# B&R Automation Studio project OpcUaSample410_BrbLibUa103 (part 2)

### RevHistory.txt
```
Revisionsgeschichte

2018-08-24	AS4.1
	Server:
		Task 'ServerData':
			-Bereitstellen von teilweisen sich ändernden Variablen über den OpcUa-Server
			-Bereistellen von Variablen, auf die die Clients schreiben können
	Client:
		Task 'ClientC' und 'ClientST':
			-Aufbauen einer Verbindung
			-Ermitteln des NamespaceIndex
			-Erzeugen von 3 Subscriptions mit MonitoredItems
			-Zyklisches Lesen einer Variablen-Liste
			-Zyklisches Schreiben einer Variablen-Liste
			-Ermitteln und Auswerten des ConnectiosStatus
			-Abbauen der Verbindung im Exit

2018-08-24	AS4.2
	Allgemein:
		-Verwendung des Rollen/Benutzer-Systems für OpcUa
		-Verwendung eines eigenen Zertifikats (Laufzeit 99 Jahre) für Server und Client
	Client:
		Task 'ClientC' und 'ClientST':
			-Hinzufügen der MonitoredItems über 'UA_MonitoredItemAddList' statt 'UA_MonitoredItemAdd'

2018-08-24	AS4.3
	Server:
		Task 'SrvMethC' und 'SrvMethST'
			-Implementierung der Methode 'Calculate'
	Client:
		Task 'ClientC' und 'ClientST':
			-Zyklischer Aufruf der Methode 'Calculate'

2018-08-24	AS4.4
	OpcUaAny:
		-Implementierung des HW-Clients, welcher nicht programmiert, sondern nur parametriert werden muss.

2018-11-19	AS4.1, AS4.2, AS4.3, AS4.4
	Client:
		Task 'ClientC' und 'ClientST':
			Das Releasen der Node-Handles, welche für die Subscription benötigt werden,
			wurde aus der Schrittkette entfernt.
			Hintergrund: Wurde die Verbindung unterbrochen und wieder hergestellt, so wurden
			die empfangenen Werte nicht mehr auf die gemappten Variablen geschrieben.
			Grundsätzlich sollten Handles nicht gelöscht werden, solange die Funktion
			benötigt wird, für die sie ermittelt wurden.

2018-11-21	AS4.4.6.71
	Server
		Task 'SrvMethC' und 'SrvMethST':
			Das ursprüngliche Projekt 'OpcUaSample44' ist aufgrund eines Fehlers in AS4.4.6.71
			nicht kompilierbar (Fehlernummer 5091), sondern nur mit AS4.4.5.61. Dehalb wurde ein
			eigenes Beispiel-Projekt 'OpcUaSample44_671' erzeugt, welches diesen Fehler umgeht.
			Hintergrund: Auf Methoden-Argumente gemappte Variablen dürfen sich in dieser Version
			nur maximal auf der 1. Ebene einer Struktur befinden, aber nicht wie im Original auf
			der 2. oder einer höheren Ebene.
			Der Fehler im AS wird schnellstmöglich (wahrscheinlich durch ein neues Upgrade)
			behoben werden.

2019-06-07	AS4.4.7.144
	Server
		Task 'SrvMethC' und 'SrvMethST':
			Der Fehler aus AS4.4.6.71 (siehe oben) wurde in dieser Version behoben. Daher wurde
			wieder auf das ursprüngliche Projekt 'OpcUaSample44' gewechselt und unter
			'OpcUaSample44_7144' abgespeichert.

2019-01-09	AS4.5
	Selbe Version wie AS4.4
		Der Fehler von '2018-11-21	AS4.4.6.71' wurde im AS behoben. Nun können auch wieder Variablen
		auf Methoden-Argumente gemappt werden, welche sich auf einer höheren Struktur-Ebene als 1 befinden.
	Überarbeitung einiger 'ReadMe.txt'-Dateien.

2019-07-05	AS4.6
	Server
		Task 'ServerData':
			Beispiele für dynamische Arrays implementiert: ByteStringExample, ByteStringExample20 und DynamicStructArray.
		Tasks 'SrvEvntC' und 'SrvEvntST':
			Beispiel zum anwenderseitigen Feuern eines Events.
		Textsystem: Sprachübersetzung des Attributs 'Description' bei den Knoten 'gVarsGlobal' und 'VarsLocal'.
	Client:
		Task 'ClientC' und 'ClientST':
			Es wurde eine Subscription implementiert, welche das Empfangen der vom Server gefeuerten Events zeigt.
	UaCerts:
		Tasks 'UaCertsC' und 'UaCertsST':
			Hier wird demonstriert, wie OpcUa-Zertifikate zur Laufzeit verwaltet werden können.

2019-07-22	AS4.6 (Eigenes Daten-Modell)
	Server
		Task 'AirCond':
			Implementierung von 3 Klima-Anlagen-Instanzen, welche über ein eigenes Modell veröffentlicht werden.
			Die Modellierung wurde komplett im externen Tool UaModeler vorgenommen.

2019-09-20	AS4.7
	AirCond (eigenes Modell):
		Es wurde ein komplett neues eigenes Modell modelliert. Die Strukturierung der Daten wurde beibehalten,
		nur deren Parametrierung wurde geändert.
		Ausserdem wurden die Vorwärts-Referenzen im externen Modell nicht mehr eingefügt. Das Mapping geschieht jetzt
		durch	Rückwärts-Referenzen, welche im AS gesetzt werden.
		Weil die Vorwärts-Referenzen auf das B&R-Modell nicht mehr nötig sind, brauchte auch das B&R-Modell nicht
		mehr ins Ua-Modeler-Projekt des eigenen Modells rückimportiert werden.
		Zusätzlich wurde ein Event 'AirConditionOperationModeChanged' implementiert. Es ist beim Knoten 'Server' und
		am Knoten der jeweiligen Instanz abgreifbar und wird immer gefeuert, wenn sich der Betriebs-Modus ändert.
	OpcUaAny:
		Durch die Verwendung eines externen Modells verschiebt sich der Namespace-Index des B&R-Modells von 6
		auf 7. Dies musste also auch in den Browse-Pfaden der OpcUaAny-Konfiguration geändert werden.
		Bei allen anderen Tasks muss nichts geändert werden, da sich diese den Namespace-Index auf das B&R-Modell
		vom Server holen.
		Leider tritt ab As4.7 + A4.73 sporadisch ein Reboot der ArSim auf, wenn im HW-Baum das Gerät 'OpcUa_any'
		aktiviert ist. Dieser Fehler ist leider noch nicht identifiziert. Daher ist das Gerät in dieser Version
		deaktiviert. Wer an dem Beispiel interessiert ist, kann das Gerät aktivieren (der Fehler tritt nicht immer
		auf). Sollte dies nicht funktionieren, kann auch mit einem älteren Beispiel gearbeitet werden, z.B. OpcUaSample46.
	ServerData:
		Das Beispiel für dynamische Arrays wurde komplett überarbeitet. Die bisherigen Beispiele wurden eliminiert und
		dafür neue implementiert, um den Unterschied zwischen 'UAArrayLength' und 'UANoOfElements' besser zu
		demonstrieren.
		Außerdem wurde die Variable 'nWritableAttributes' implementiert, um die Funktionalität 'Schreibbare Attribute'
		zu zeigen.

Hinweis zu AS4.8
	Es gibt kein Sample48, da in dieser Version keine nennenswerten neuen Funktionalitäten hinzugekommen sind.
	Es wurden nur Fehler- und Performance-Optimierungen im AS und AR gemacht.

2021-03-25	AS4.9
	Erweiterung um ein Publisher/Subscriber-Beispiel.
		Es wurde sowohl ein Publisher als auch Subscriber konfiguriert, welche zusammen passen. Auch die programmseitige
		Diagnose mittels Zähler wird demonstriert.
	Fehler in FireEvent (Task 'SrvEvent')
		Leider hat sich in der verwendeten Betriebssystem-Version A4.90 ein Fehler eingesschlichen. Wird am Field 'Context'
		eine Struktur-Variable angebunden, deren Struktur-Definition global angelegt ist (wie es legitim ist und normalerweise
		in diesem Beispiel gezeigt wird), so liefert der FB den Fehler 0x803D0000 = 'Bad_NotSupported' zurück, statt das Event zu
		feuern. Daher ist für diese Version	lediglich ein REAL angebunden. Sobald der Fehler in einer der nächsten Versionen
		behoben ist, wird das Beispiel wieder eine Struktur anbinden.

2021-09-14	As4.9 (BrbLibUa)
	Umstellung von AR A4.90 auf E4.90.
	Fehler in FireEvent (Task 'SrvEvent') ist behoben.
		Der oben beschriebene Fehler zum Field 'Context' (globale Definition der Struktur) wurde in E4.90 behoben. Daher wird hier
		auch wieder die Struktur angebunden (siehe ServerEvents\ReadMe.txt).
	Erweiterung um Bibliothek 'BrbLibUa' und deren Beispiele.
		Hier wird gezeigt, wie mithilfe dieser Bibliothek viele Funktionalitäten von Server und Client implementiert werden
		können. Im Gegensatz zur herkömmlichen Programmierung ist dann sehr viel weniger Aufwand nötig.
	Eliminierung der Hilfs-Bibliothek 'Util'
		Da alle benötigten Funktionen dieser Hilfs-Bibliothek in der Bibliothek 'BrbLib' vorhanden sind und diese sowieso
		für die 'BrbLibUa' gebraucht wird, wurde 'Util' entfernt.

2022-05-13	As4.10  (BrbLibUa V1.01)
	Umstellung von AR E4.90 auf D4.91.
	BrbLibUa V1.01 (genaueres zu Erweiterungen/Korrekturen siehe Dokumentation der Bibliothek)
	Task 'BrbUaClt': Die neue Funktion BrbUaGetSrvTimeText() wird beispielhaft verwendet.

2022-06-07	As4.10 (BrbLibUa V1.02)
	BrbLibUa V1.02 (genaueres zu Erweiterungen/Korrekturen siehe Dokumentation der Bibliothek).
	Implementierung der UnitTests für BrbLibUa.
	Die Compiler-Version wurde von V4.1.2 auf 6.3.0 geändert.
	Die Abhängigkeit von der Basis-Bibliothek 'BrbLib' wurde von V5.01 auf V5.02 geändert.
	Prüfung mit dem Code-Analyse-Tool 'ClangTidy'. Dies führt zu einer erhöhten SW-Qualität.
	Server
		Task 'SrvDt64C' und 'SrvDt64ST':
			Implementierung von 64-Bit-Datentypen wie Uint64 (ULINT) und Int64 (LINT).
	Client
		Task 'BrbUaClient': Abonnieren der Server-Info- und Server-Diagnose-Daten beispielhaft implementiert.

2024-02-22	As4.10 (BrbLibUa V1.03)
	Umstellung von AR E4.91 auf H4.91.
	Die Bibliothek BrbLib wurde von V5.02 auf V5.03 upgedatet (genaueres zu Erweiterungen/Korrekturen siehe Dokumentation der Bibliothek).
	BrbLibUa V1.03:
		Die Abhängigkeit zur Bibliothek 'BrbLib' wurde von V5.02 auf V50.3 erhöht.
		Es wurden Hinweise in die Hilfe aufgenommen.
		Die Bibliothek selbst hat sich nicht geändert.
	Prüfung mit neuer Version des Code-Analyse-Tools 'ClangTidy'. Dies führt zu einer erhöhten SW-Qualität.
	ServerEvents: Die Variable 'Fields.nSeverity' war fälschlicherweise als INT deklariert. Jetzt ist es korrekt ein UINT.
	Korrektur in den Client-Tasks 'ClientC' und 'ClientST': In folgenden Schritten wurden bei FB-Fehlermeldungen die ErrorID vom falschen
		FB übernommen: eSTEP_CREATE_SUBSCRIPT_VAR_WAIT, eSTEP_CREATE_SUBSCRIPT_EVT_WAIT.
		Dies ist jetzt korrigiert.
	ClientC und ClientST: Hinweis aufgenommen, dass zyklisches Lesen (Polling) niemals in einer Applikation implementiert werden sollte.
```

### ReadMe.txt
```
In diesem Beispiel wird die Implementierung von OpcUa-Funktionalitäten gezeigt.
Es ist KEIN offizielles Beispiel und daher besteht für den Anwender kein Anspruch auf
Erweiterung, Fehlerbehebung, Schulung oder Support. Auch die Fehlerfreiheit kann nicht
garantiert werden.

Tasks
	Template:				Ist ein Muster, um schneller neue Tasks im selben Format implementieren zu können.
									Es wird für das Beispiel nicht benötigt.
	ServerData: 		Stellt Variablen zur Verfügung, die am eigenen Server veröffentlicht werden und Variablen, welche
									von den Clients beschrieben werden.
	SrvDt64C:				Die Implementierung von 64-Bit-Werten in der Sprache ANSI-C;
	SrvDt64ST:			Die Implementierung von 64-Bit-Werten in der Sprache StructuredText;
	SrvMethC:				Die Implementierung benutzerdefinierten Server-Methoden in der Sprache ANSI-C.
	SrvMethST:			Die Implementierung benutzerdefinierten Server-Methoden in der Sprache StructuredText.
	SrvEvntC:				Anwenderseitiges Feuern eines Events in der Sprache ANSI-C.
	SrvEvntST:			Anwenderseitiges Feuern eines Events in der Sprache StructuredText. Dieser Task ist disabled.
	ClientC:				Die Implementierung des Clients in der Sprache ANSI-C.
	ClientST:				Die Implementierung des Clients in der Sprache StructuredText.
	BrbUaCltC:			Die Implementierung des Clients mithilfe der Bibiothk BrbLibUa in der Sprache ANSI-C.
	BrbUaCltST:			Die Implementierung des Clients mithilfe der Bibiothk BrbLibUa in der StructuredText.
	OpcUaAny:				Stellt lediglich Variablen bereit, welche am OpcUaAny-Client gemappt sind.
	BrbUaSrvC:			Die Implementierung des Servers mithilfe der Bibiothk BrbLibUa in der Sprache ANSI-C.
	BrbUaSrvST:			Die Implementierung des Servers mithilfe der Bibiothk BrbLibUa in der StructuredText.
	UaCertsC:				Beispiel zur Laufzeit-Verwaltung von Zertifikaten in der Sprache ANSI-C.
	UaCertsST:			Beispiel zur Laufzeit-Verwaltung von Zertifikaten in der Sprache StructuredText.
	AirCondC:				Funktionelle Implementierung für das Beispiel eines eigenen Datenmodells in der Sprache ANSI-C.
	AirCondST:			Funktionelle Implementierung für das Beispiel eines eigenen Datenmodells in der Sprache StructuredText.
	PubSub:					Exemplarische Konfiguration einer PubSub-Verbindung.

In jedem Task ist ebenfalls eine ReadMe.txt enthalten, die ihn näher beschreibt.
Der Task 'SrvEvntST' ist disabled, damit das Event nicht vom ANSIC- und vom ST-Task gefeuert wird.

Um dieses Beispiel zu verstehen, ist es zwingend notwendig, die AS-Hilfe zu studieren. Ausserdem sollte sich der
Anwender Wissen über Konzepte und die allgemeine Funktionsweise von OpcUa aneignen. B&R bietet hierfür auch Kurse an.

Ab AS4.4 kann als Ersatz für den Library-Client der OpcUa_Any-Client verwendet werden, welcher im HW-Baum
eingefügt wird und nur parametriert statt programmiert werden muss.

Ab AS4.9 kann ein Library-Client mit sehr viel weniger Aufwand mithilfe der Bibliothek BrbLibUa implementiert werden.
Auch hier ist ein Beispiel vorhanden.

WICHTIG:
Wird kein jeweils eigenes Zertifikat für Server/Client angelegt, werden beim erstmaligem Starten der SPS
automatisch Zertifikate erzeugt, welche aber nur einen Gültigkeitszeitraum von 10 Jahren haben.
Bei einer Verbindung zwischen B&R-Teilnehmern ist das unkritisch, da dann der Gültigkeitszeitraum nicht
geprüft wird. Bei einer Verbindung zu einem externen Teilnehmer (also nicht B&R) muss ermittelt werden, ob
dieser den Gültigkeitszeitraum prüft und gegebenenfalls eine Verbindugn zurückweist!
Ist das der Fall, sollten also unbedingt eigene Zertifikate angelegt und verwendet werden.
Siehe dazu AS-Hilfe GUID 'f83f9b82-60fe-4f7c-b101-504cb81ffc44' (='Access & Security/TLS/SSL(SSL bei B&R') sowie
GUID '2c919423-08bb-4895-88b8-afcf6114d0a2' (='Programmierung/Editoren/Konfigurationseditoren/
Hardwarekonfiguration/CPU Konfiguration/SG4/OPC UA Server').
In diesem Beispiel wurde jeweils ein Zertifikat für Server und Client unter
'ConfigurationView/AccessAndSecurity/CertificateStore/OwnCertifcates' mit einer Laufzeit von 50 Jahren
angelegt.
Dazu wurde die Konfiguration 'ConfigurationView/AccessAndSecurity/TransortLayerSecurity/OpcUaCfg.sslcfg'
angelegt, in welcher die Einträge konfiguriert sind.
Die Konfiguration 'SslCfgOpcUaServer' wurde dem Server in der System-Konfiguration zugewiesen.
Die Konfiguration 'SslCfgOpcUaClient' wird dem Client am FB 'UA_Connect' zugewiesen.
Siehe dazu auch Package 'UACerts'.
```

### Global.typ - Global data types
```iecst
TYPE
	OpcUaTestDatatypes_TYP : 	STRUCT
		bBool : BOOL;
		nUsint : USINT;
		nUint : UINT;
		nUdint : UDINT;
		nSint : SINT;
		nInt : INT;
		nDint : DINT;
		rReal : REAL;
		rLongReal : LREAL;
		sString : STRING[nOPCUA_STRING_CHAR_MAX];
		tTime : TIME;
		dtDateTime : DATE_AND_TIME;
		anInt : ARRAY[0..nOPCUA_ARRAY_INDEX_MAX]OF INT;
	END_STRUCT;
	OpcUaServerVars_TYP : 	STRUCT
		WriteOnly : OpcUaTestDatatypes_TYP;
		ReadOnly : OpcUaTestDatatypes_TYP;
		ReadWrite : OpcUaTestDatatypes_TYP;
	END_STRUCT;
	ClientCfgConnectionTYP : 	STRUCT
		UserIdentityToken : UAUserIdentityToken;
		tSessionTimeout : TIME;
		tMonitorConnection : TIME;
		sServerEndpointUrl : STRING[nENDPOINT_URL_CHAR_MAX];
	END_STRUCT;
	ClientCfgSubscriptionsTYP : 	STRUCT
		sNamespaceUriOrg : STRING[nNAMESPACE_URI_CHAR_MAX];
		nNamespaceUriOrg : UINT;
		sNamespaceUriBrPv : STRING[nNAMESPACE_URI_CHAR_MAX];
		nNamespaceUriBrPv : UINT;
		SubVar : ARRAY[0..nCLIENT_SUBSCRIPTION_INDEX_MAX]OF ClientCfgSubscriptionVarTYP;
		SubEvt : ClientCfgSubscriptionEvtTYP;
	END_STRUCT;
	ClientCfgSubscriptionVarTYP : 	STRUCT
		tPublishingInterval : TIME;
		nPriority : BYTE;
		MonitoredItem : ARRAY[0..nCLIENT_MONITORED_ITEM_INDEX_MAX]OF ClientCfgMonItemTYP;
	END_STRUCT;
	ClientCfgMonItemTYP : 	STRUCT
		NodeId : UANodeID;
		sVarName : STRING[nVAR_NAME_CHAR_MAX];
	END_STRUCT;
	ClientCfgSubscriptionEvtTYP : 	STRUCT
		tPublishingInterval : TIME;
		nPriority : BYTE;
		NotifierNodeId : UANodeID;
		EventTypeNodeId : UANodeID;
		EventFieldVarNames : ARRAY[0..MAX_INDEX_EVENTFIELDSELECTION]OF STRING[MAX_LENGTH_VARIABLE];
	END_STRUCT;
	ClientCfgReadTYP : 	STRUCT
		Item : ARRAY[0..nCLIENT_READ_ITEM_INDEX_MAX]OF ClientCfgMonItemTYP;
	END_STRUCT;
	ClientCfgWriteTYP : 	STRUCT
		Item : ARRAY[0..nCLIENT_WRITE_ITEM_INDEX_MAX]OF ClientCfgMonItemTYP;
	END_STRUCT;
	ClientCfgMethodsTYP : 	STRUCT
		Method : ARRAY[0..nCLIENT_METHODS_INDEX_MAX]OF ClientCfgMethodTYP;
	END_STRUCT;
	ClientCfgMethodTYP : 	STRUCT
		ObjectNodeId : UANodeID;
		MethodNodeId : UANodeID;
		ArgumentsIn : ARRAY[0..MAX_INDEX_ARGUMENTS]OF UAMethodArgument;
		ArgumentsOut : ARRAY[0..MAX_INDEX_ARGUMENTS]OF UAMethodArgument;
	END_STRUCT;
	ClientCfgTYP : 	STRUCT
		Connection : ClientCfgConnectionTYP;
		Subscriptions : ClientCfgSubscriptionsTYP;
		Read : ClientCfgReadTYP;
		Write : ClientCfgWriteTYP;
		Methods : ClientCfgMethodsTYP;
	END_STRUCT;
	ClientConnectionStatus_TYP : 	STRUCT
		eConnectionStatus : UAConnectionStatus;
		eServerState : UAServerState;
		eServerLevel : BYTE;
	END_STRUCT;
	MethCalculateArgsIn_TYP : 	STRUCT
		nVal0 : DINT;
		nVal1 : DINT;
		anArray : ARRAY[0..nMETHOD_CALC_ARRAY_INDEX_MAX]OF INT;
	END_STRUCT;
	MethCalculateArgsOut_TYP : 	STRUCT
		nAddition : DINT;
		nMultiplication : DINT;
		anArray : ARRAY[0..nMETHOD_CALC_ARRAY_INDEX_MAX]OF INT;
	END_STRUCT;
	MethCalculateArgs_TYP : 	STRUCT
		In : MethCalculateArgsIn_TYP;
		Out : MethCalculateArgsOut_TYP;
	END_STRUCT;
	EventFieldContext_TYP : 	STRUCT
		nUsint : USINT;
		rReal : REAL;
		sString : STRING[255];
	END_STRUCT;
	ClientReceivedMonItem_TYP : 	STRUCT
		bValueChanged : BOOL;
		nReceivedCount : UDINT;
	END_STRUCT;
	ProgressEvent_TYP : 	STRUCT
		nReceivedCount : UDINT;
		EventId : UAByteStringBrbEventId_TYP;
		sEventIdHex : STRING[255];
		EventType : UANodeID;
		LocalTime : UATimeZoneData;
		Message : UALocalizedText;
		ReceiveTime : UaSrv_DateTimeType;
		Severity : UINT;
		SourceName : STRING[nBRBUA_VALUE_TEXT_CHAR_MAX];
		SourceNode : UANodeID;
		Time : UaSrv_DateTimeType;
		Context : EventFieldContext_TYP;
		Progress : UINT;
	END_STRUCT;
	TransitionEvent_TYP : 	STRUCT
		nReceivedCount : UDINT;
		EventId : UAByteStringBrbEventId_TYP;
		sEventIdHex : STRING[255];
		EventType : UANodeID;
		LocalTime : UATimeZoneData;
		Message : UALocalizedText;
		ReceiveTime : UaSrv_DateTimeType;
		sReceiveTime : STRING[64];
		nSeverity : UINT;
		sSourceName : STRING[nBRBUA_VALUE_TEXT_CHAR_MAX];
		SourceNode : UANodeID;
		FromState : UALocalizedText;
		nFromStateId : UINT;
		ToState : UALocalizedText;
		nToStateId : UINT;
		Transition : UALocalizedText;
		nTransitionId : DINT;
	END_STRUCT;
	PubSubDiagDataMsg_TYP : 	STRUCT
		nTotal : UDINT;
		nError : UDINT;
	END_STRUCT;
	PubSubDiagData_TYP : 	STRUCT
		UdpMessage : PubSubDiagDataMsg_TYP;
		DataSet : PubSubDiagDataMsg_TYP;
	END_STRUCT;
END_TYPE
```

### Global.var - Global variables
```iecst
VAR CONSTANT
	nSTEP_TEXT_CHAR_MAX : UINT := 100;
	nOPCUA_STRING_CHAR_MAX : UINT := 255;
	nOPCUA_ARRAY_INDEX_MAX : UINT := 4;
	tFB_TIMEOUT : TIME := T#2s;
	nENDPOINT_URL_CHAR_MAX : UINT := 255;
	nNAMESPACE_URI_CHAR_MAX : UINT := 255;
	nCLIENT_SUBSCRIPTION_INDEX_MAX : UINT := 2;
	nCLIENT_MONITORED_ITEM_INDEX_MAX : UINT := 3;
	nCLIENT_READ_ITEM_INDEX_MAX : UINT := 2;
	nCLIENT_WRITE_ITEM_INDEX_MAX : UINT := 2;
	nCLIENT_METHODS_INDEX_MAX : UINT := 0;
	nVAR_NAME_CHAR_MAX : UINT := 255;
	nMETHOD_CALC_ARRAY_INDEX_MAX : UINT := 3;
END_VAR
```

### Package Logical/Libraries - Global libraries

### Library Logical/Libraries/BrbLib (ANSIC, version 5.03.0) - Helpful functions
Depends on: standard, astime, AsBrStr, FileIO, sys_lib, DataObj, AsUSB, AsBrWStr, ArEventLog

#### BrbLib.fun - Exported functions and function blocks
```iecst
(********************************************************************
 * COPYRIGHT -- Bernecker + Rainer
 ********************************************************************
 * Library: BrbLib
 * File: BrbLib.fun
 * Author: niedermeierr
 * Created: June 11, 2013
 ********************************************************************
 * Functions and function blocks of library BrbLib
 ********************************************************************)
(*StepHandling*)

FUNCTION BrbStepHandler : DINT (*Behandelt Schrittketten (Protokollierung, Timeout usw.)*)
	VAR_INPUT
		pStepHandling : BrbStepHandling_TYP; (*Zeiger auf eine lokale Struktur "BrbStepHandling_TYP"*)
	END_VAR
END_FUNCTION

FUNCTION BrbStartStepTimeout : UINT (*Startet den Timeout-Zähler für eine Schrittkette*)
	VAR_INPUT
		pStepHandling : BrbStepHandling_TYP; (*Zeiger auf eine lokale Struktur "BrbStepHandling_TYP"*)
		nTimeout : UDINT; (*Zeitangabe in [ms]*)
		nContinueStep : DINT; (*Schrittnummer bei abgelaufenem Timeout*)
	END_VAR
END_FUNCTION

FUNCTION BrbStopStepTimeout : UINT (*Stoppt den Timeout-Zähler für eine Schrittkette*)
	VAR_INPUT
		pStepHandling : BrbStepHandling_TYP; (*Zeiger auf eine lokale Struktur "BrbStepHandling_TYP"*)
	END_VAR
END_FUNCTION

FUNCTION BrbStartStopWatch : BOOL (*Startet eine Stoppuhr*)
	VAR_INPUT
		pStopWatch : BrbStopWatch_TYP; (*Zeiger auf eine lokale Struktur "BrbStopWatch_TYP"*)
	END_VAR
END_FUNCTION

FUNCTION BrbStopStopWatch : UDINT (*Stoppt eine Stoppuhr*)
	VAR_INPUT
		pStopWatch : BrbStopWatch_TYP; (*Zeiger auf eine lokale Struktur "BrbStopWatch_TYP"*)
	END_VAR
END_FUNCTION
(*TaskCommunication*)

FUNCTION BrbSetCaller : BrbCallerStates_ENUM (*Versucht, die Reservierung für ein Task-Kommando zu erhalten*)
	VAR_INPUT
		pCaller : BrbCaller_TYP; (*Zeiger auf eine Struktur "BrbCaller_TYP"*)
		nCallerId : DINT; (*Identifier für den aufrufenden Task*)
	END_VAR
END_FUNCTION

FUNCTION BrbClearDirectBox : UINT (*Setzt eine DirectBox komplett auf 0*)
	VAR_INPUT
		pDirectBox : UDINT; (*Zeiger auf eine DirectBox-Struktur*)
		nSize : UDINT; (*Größe der Struktur*)
	END_VAR
END_FUNCTION

FUNCTION BrbClearCallerBox : UINT (*Setzt eine CallerBox komplett auf 0*)
	VAR_INPUT
		pCallerBox : UDINT; (*Zeiger auf eine CallerBox-Struktur*)
		nSize : UDINT; (*Größe der Struktur*)
	END_VAR
END_FUNCTION
(*VarHandling*)

{REDUND_UNREPLICABLE} FUNCTION_BLOCK BrbSaveVarAscii (*Speichert eine Variable mit allen Elementen in einer Ascii-Datei*)
	VAR_INPUT
		pDevice : REFERENCE TO STRING[0]; (*Zeiger auf den Laufwerks-Namen*)
		pFile : REFERENCE TO STRING[0]; (*Zeiger auf den Datei-Namen*)
		pVarName : REFERENCE TO STRING[0]; (*Zeiger auf den Variablen-Namen*)
		nLinesToWriteAtOneStep : {REDUND_UNREPLICABLE} UINT; (*Anzahl der Zeilen, die in einem Aufruf geschrieben werden*)
	END_VAR
	VAR_OUTPUT
		nCharCountMaxPerWrite : {REDUND_UNREPLICABLE} UDINT; (*Größte Anzahl der Zeichen, welche in einer Zeile geschrieben wurden*)
		nStatus : {REDUND_UNREPLICABLE} UINT; (*Fub-Status*)
	END_VAR
	VAR
		eStep : {REDUND_UNREPLICABLE} DINT; (*Step-Nummer für die interne Schrittkette*)
		nStatusIntern : {REDUND_UNREPLICABLE} UINT; (*Interner Fub-Status*)
		fbFileDelete : {REDUND_UNREPLICABLE} FileDelete; (*Fub zum Löschen der Datei*)
		fbFileCreate : {REDUND_UNREPLICABLE} FileCreate; (*Fub zum Erzeugen der Datei*)
		sHelp : {REDUND_UNREPLICABLE} STRING[nBRB_PVNAME_CHAR_MAX]; (*Hilfsstring*)
		nOffset : {REDUND_UNREPLICABLE} UDINT; (*Schreib-Offset*)
		nLineCountWrite : {REDUND_UNREPLICABLE} UDINT; (*Zeilen-Zähler*)
		bVarFinished : {REDUND_UNREPLICABLE} BOOL; (*1= Variable komplett durchgetickert*)
		PvInfo : {REDUND_UNREPLICABLE} ARRAY[0..16] OF BrbPvInfo_TYP; (*Struktur für Variablen-Daten*)
		nPvLevel : {REDUND_UNREPLICABLE} UINT; (*Hierarchie-Level für Strukturen*)
		sLines : {REDUND_UNREPLICABLE} STRING[nBRB_FILE_LINES_CHAR_MAX]; (*Text-Zeilen*)
		fbFileWrite : {REDUND_UNREPLICABLE} FileWrite; (*Fub zum Schreiben der Datei*)
		fbFileClose : {REDUND_UNREPLICABLE} FileClose; (*Fub zum Schliessen der Datei*)
	END_VAR
END_FUNCTION_BLOCK

FUNCTION_BLOCK BrbLoadVarAscii (*Lädt eine Ascii-Datei mit Variablen-Werten*)
	VAR_INPUT
		pDevice : REFERENCE TO STRING[0]; (*Zeiger auf den Laufwerks-Namen*)
		pFile : REFERENCE TO STRING[0]; (*Zeiger auf den Datei-Namen*)
		eLineBeak : BrbLineBreak_ENUM; (*Verwendeter Zeilenumbruch*)
		nLinesToReadAtOneStep : {REDUND_UNREPLICABLE} UINT; (*Anzahl der Zeilen, die in einem Aufruf gelesen werden*)
	END_VAR
	VAR_OUTPUT
		nStatus : {REDUND_UNREPLICABLE} UINT; (*Fub-Status*)
	END_VAR
	VAR
		eStep : {REDUND_UNREPLICABLE} DINT; (*Step-Nummer für die interne Schrittkette*)
		nStatusIntern : {REDUND_UNREPLICABLE} UINT; (*Interner Fub-Status*)
		fbDatObjInfo : {REDUND_UNREPLICABLE} DatObjInfo; (*Fub zum Holen der Datenobjekt-Info*)
		fbFileOpen : {REDUND_UNREPLICABLE} FileOpen; (*Fub zum Öffnen der Datei*)
		fbDatObjCreate : {REDUND_UNREPLICABLE} DatObjCreate; (*Fub zum Erzeugen des Datenobjekts*)
		sLineBreak : STRING[8]; (*Verwendeter Zeilenumbruch*)
		pTextStart : REFERENCE TO STRING[0]; (*Zeiger auf den Anfang des eingelesenen Texts*)
		pTextEnd : REFERENCE TO STRING[0]; (*Zeiger auf das Ende des eingelesenen Texts*)
		pText : REFERENCE TO STRING[0]; (*Zeiger auf den aktuellen Text*)
		nLineCountRead : {REDUND_UNREPLICABLE} UDINT; (*Anzahl der eingelesenen Zeilen*)
		fbFileRead : {REDUND_UNREPLICABLE} FileRead; (*Fub zum Lesen der Datei*)
		fbFileClose : {REDUND_UNREPLICABLE} FileClose; (*Fub zum Schliessen der Datei*)
		fbDatObjDelete : {REDUND_UNREPLICABLE} DatObjDelete; (*Fub zum Löschen des Datenobjekts*)
	END_VAR
END_FUNCTION_BLOCK

{REDUND_UNREPLICABLE} FUNCTION_BLOCK BrbSaveVarBin (*Speichert eine Variable mit allen Elementen in einer Binär-Datei*)
	VAR_INPUT
		pDevice : REFERENCE TO STRING[0]; (*Zeiger auf den Laufwerks-Namen*)
		pFile : REFERENCE TO STRING[0]; (*Zeiger auf den Datei-Namen*)
		pVarName : REFERENCE TO STRING[0]; (*Zeiger auf den Variablen-Namen*)
	END_VAR
	VAR_OUTPUT
		nStatus : {REDUND_UNREPLICABLE} UINT; (*Fub-Status*)
	END_VAR
	VAR
		eStep : {REDUND_UNREPLICABLE} DINT; (*Step-Nummer für die interne Schrittkette*)
		nStatusIntern : {REDUND_UNREPLICABLE} UINT; (*Interner Fub-Status*)
		PvInfo : {REDUND_UNREPLICABLE} BrbPvInfo_TYP; (*Struktur für Variablen-Daten*)
		fbFileDelete : {REDUND_UNREPLICABLE} FileDelete; (*Fub zum Löschen der Datei*)
		fbFileCreate : {REDUND_UNREPLICABLE} FileCreate; (*Fub zum Erzeugen der Datei*)
		fbFileWrite : {REDUND_UNREPLICABLE} FileWrite; (*Fub zum Schreiben der Datei*)
		fbFileClose : {REDUND_UNREPLICABLE} FileClose; (*Fub zum Schliessen der Datei*)
	END_VAR
END_FUNCTION_BLOCK

{REDUND_UNREPLICABLE} FUNCTION_BLOCK BrbLoadVarBin (*Lädt eine Binär-Datei mit Variablen-Werten*)
	VAR_INPUT
		pDevice : REFERENCE TO STRING[0]; (*Zeiger auf den Laufwerks-Namen*)
		pFile : REFERENCE TO STRING[0]; (*Zeiger auf den Datei-Namen*)
		pVarName : REFERENCE TO STRING[0]; (*Zeiger auf den Variablen-Namen*)
		bAllowBiggerVar : {REDUND_UNREPLICABLE} BOOL; (*1=Der Speicher der Variablen darf größer als die Datei sein*)
	END_VAR
	VAR_OUTPUT
		nStatus : {REDUND_UNREPLICABLE} UINT; (*Fub-Status*)
	END_VAR
	VAR
		eStep : {REDUND_UNREPLICABLE} DINT; (*Step-Nummer für die interne Schrittkette*)
		nStatusIntern : {REDUND_UNREPLICABLE} UINT; (*Interner Fub-Status*)
		fbFileOpen : {REDUND_UNREPLICABLE} FileOpen; (*Fub zum Öffnen der Datei*)
		PvInfo : {REDUND_UNREPLICABLE} BrbPvInfo_TYP; (*Struktur für Variablen-Daten*)
		fbFileRead : {REDUND_UNREPLICABLE} FileRead; (*Fub zum Lesen der Datei*)
		fbFileClose : {REDUND_UNREPLICABLE} FileClose; (*Fub zum Schliessen der Datei*)
	END_VAR
END_FUNCTION_BLOCK
(*FileHandling*)

{REDUND_UNREPLICABLE} FUNCTION_BLOCK BrbReadDir (*Gibt eine Liste der Dateien und/oder der Verzeichnisse eines Laufwerks zurück*)
	VAR_INPUT
		pDevice : REFERENCE TO STRING[0]; (*Zeiger auf den Laufwerks-Namen*)
		pPath : REFERENCE TO STRING[0]; (*Zeiger auf den Pfad*)
		eFilter : {REDUND_UNREPLICABLE} BrbDirInfoFilter_ENUM; (*Datei- und Verzeichnis-Filter*)
		bWithParentDir : {REDUND_UNREPLICABLE} BOOL; (*1=Mit übergeordnetem Verzeichnis*)
		pFileFilter : REFERENCE TO STRING[0]; (*Zeiger auf den Filtertext für Datei-Endungen*)
		bUserFilter : {REDUND_UNREPLICABLE} BOOL; (*1=Benutzerdefinierte Filterfunktion wird zusätzlich verwendet*)
		pUserFilterFunction : {REDUND_UNREPLICABLE} UDINT; (*Zeiger auf die benutzerdefinierte Filterfunktion*)
		eSorting : {REDUND_UNREPLICABLE} BrbFileSorting_ENUM; (*Sortierung*)
		bCaseSensitive : {REDUND_UNREPLICABLE} BOOL; (*1=Groß-/Klein-Schreibung beachten (gitl nur bei alphanumerischer Sortierung)*)
		pUserCompareFunction : {REDUND_UNREPLICABLE} UDINT; (*Zeiger auf die benutzerdefinierte Vergleichsfunktion bei 'eBRB_FILE_SORTING_USER'*)
		pList : {REDUND_UNREPLICABLE} UDINT; (*Zeiger auf das zu füllende Array*)
		nListIndexMax : {REDUND_UNREPLICABLE} UDINT; (*Maximaler Anzahl der Einträge im Array*)
	END_VAR
	VAR_OUTPUT
		nDirCount : {REDUND_UNREPLICABLE} UDINT; (*Anzahl der Verzeichnisse in der Liste*)
		nFileCount : {REDUND_UNREPLICABLE} UDINT; (*Anzahl der Dateien in der Liste*)
		nTotalCount : {REDUND_UNREPLICABLE} UDINT; (*Anzahl der Verzeichnisse und Dateien in der Liste*)
		nStatus : {REDUND_UNREPLICABLE} UINT; (*Fub-Status*)
	END_VAR
	VAR
		eStep : {REDUND_UNREPLICABLE} DINT; (*Step-Nummer für die interne Schrittkette*)
		FilterListMan : {REDUND_UNREPLICABLE} BrbMemListManagement_Typ; (*Verwaltung der Filter-Liste*)
		FilterList : {REDUND_UNREPLICABLE} ARRAY[0..nBRB_FILTER_SINGLE_INDEX_MAX] OF STRING[nBRB_FILTER_SINGLE_CHAR_MAX]; (*Liste der Filter*)
		fbDirRead : {REDUND_UNREPLICABLE} DirRead; (*Fub zum Auslesen des Laufwerks*)
		FileInfo : {REDUND_UNREPLICABLE} fiDIR_READ_DATA; (*Daten der aktueller Datei*)
		ReadListEntry : {REDUND_UNREPLICABLE} BrbReadDirListEntry_TYP; (*Daten der aktueller Datei*)
		FileListMan : {REDUND_UNREPLICABLE} BrbMemListManagement_Typ; (*Verwaltung der Datei-Liste*)
	END_VAR
END_FUNCTION_BLOCK

{REDUND_UNREPLICABLE} FUNCTION_BLOCK BrbCheckUsbSticks (*Prüft, ob ein Usb-Stick gesteckt wurde*)
	VAR_INPUT
		bAutoLink : {REDUND_UNREPLICABLE} BOOL; (*1=Usb-Device wird beim Stecken automatisch gelinkt*)
	END_VAR
	VAR_OUTPUT
		nUsbDeviceCount : {REDUND_UNREPLICABLE} UINT; (*Anzahl der gesteckten Usb-Sticks*)
		bUsbDeviceCountChanged : {REDUND_UNREPLICABLE} BOOL; (*Anzahl hat sich geändert (nur 1 für einen Zyklus)*)
		UsbDeviceList : {REDUND_UNREPLICABLE} ARRAY[0..nBRB_USB_DEVICE_LIST_INDEX_MAX] OF BrbUsbDeviceListEntry_TYP; (*Liste der Usb-Devices*)
		nStatus : {REDUND_UNREPLICABLE} UINT; (*Fub-Status*)
	END_VAR
	VAR
		eStep : {REDUND_UNREPLICABLE} DINT; (*Step-Nummer für die interne Schrittkette*)
		DeviceListMan : {REDUND_UNREPLICABLE} BrbMemListManagement_Typ; (*Verwaltung der Device-Liste*)
		nUsbDeviceIndex : {REDUND_UNREPLICABLE} UINT; (*Aktueller Index in der Device-Liste*)
		UsbDeviceListEntry : {REDUND_UNREPLICABLE} BrbUsbDeviceListEntry_TYP; (*Aktueller Eintrag in der Device-Liste*)
		fbUsbNodeListGet : {REDUND_UNREPLICABLE} UsbNodeListGet; (*Fub zum Lesen der Node-Liste*)
		nUsbNodeIndex : {REDUND_UNREPLICABLE} UINT; (*Aktueller Index in der Node-Liste*)
		UsbNodeList : {REDUND_UNREPLICABLE} ARRAY[0..nBRB_USB_DEVICE_LIST_INDEX_MAX] OF UDINT; (*Node-Liste*)
		nAttachDetachCountOld : {REDUND_UNREPLICABLE} UDINT; (*Vergleichs-Zähler*)
		fbDevUnlink : {REDUND_UNREPLICABLE} DevUnlink; (*Fub zum Unlinken*)
		fbUsbNodeGet : {REDUND_UNREPLICABLE} UsbNodeGet; (*Fub zum Lesen der Node-Info*)
		UsbNodeInfo : {REDUND_UNREPLICABLE} usbNode_typ; (*Node-Info*)
		sLinkParameter : {REDUND_UNREPLICABLE} STRING[100]; (*Parameter zum Linken*)
		fbDevLink : {REDUND_UNREPLICABLE} DevLink; (*Fub zum Linken*)
	END_VAR
END_FUNCTION_BLOCK

{REDUND_UNREPLICABLE} FUNCTION_BLOCK BrbDeleteFiles (*Löscht Dateien, die über Filter festgelegt sind*)
	VAR_INPUT
		pDevice : REFERENCE TO STRING[0]; (*Zeiger auf den Laufwerks-Namen*)
		pPath : REFERENCE TO STRING[0]; (*Zeiger auf den Pfad*)
		pFileFilter : REFERENCE TO STRING[0]; (*Zeiger auf den Filtertext für Datei-Endungen*)
		dtDateStart : {REDUND_UNREPLICABLE} DATE_AND_TIME; (*Angabe des Start-Datums*)
		dtDateEnd : {REDUND_UNREPLICABLE} DATE_AND_TIME; (*Angabe des Ende-Datums*)
	END_VAR
	VAR_OUTPUT
		nDeletedFileCount : {REDUND_UNREPLICABLE} UDINT; (*Anzahl der gelöschten Dateien*)
		nKeptFileCount : {REDUND_UNREPLICABLE} UDINT; (*Anzahl der nicht gelöschten Dateien*)
		nStatus : {REDUND_UNREPLICABLE} UINT; (*Fub-Status*)
	END_VAR
	VAR
		eStep : {REDUND_UNREPLICABLE} DINT; (*Step-Nummer für die interne Schrittkette*)
		FilterListMan : {REDUND_UNREPLICABLE} BrbMemListManagement_Typ; (*Verwaltung der Filter-Liste*)
		FilterList : {REDUND_UNREPLICABLE} ARRAY[0..nBRB_FILTER_SINGLE_INDEX_MAX] OF STRING[nBRB_FILTER_SINGLE_CHAR_MAX]; (*Liste der Filter*)
		fbDirRead : {REDUND_UNREPLICABLE} DirRead; (*Fub zum Auslesen des Laufwerks*)
		FileInfo : {REDUND_UNREPLICABLE} fiDIR_READ_DATA; (*Daten der aktueller Datei*)
		sFileWithPath : {REDUND_UNREPLICABLE} STRING[nBRB_FILE_NAME_CHAR_MAX]; (*Pfad mit Dateiname*)
		fbFileDelete : {REDUND_UNREPLICABLE} FileDelete; (*Fub zum Auslesen des Laufwerks*)
	END_VAR
END_FUNCTION_BLOCK

{REDUND_UNREPLICABLE} FUNCTION_BLOCK BrbLoadFileDataObj (*Lädt eine Datei in ein Datenobjekt*)
	VAR_INPUT
		pDevice : REFERENCE TO STRING[0]; (*Zeiger auf den Laufwerks-Namen*)
		pFile : REFERENCE TO STRING[0]; (*Zeiger auf den Datei-Namen*)
		pDataObjName : REFERENCE TO STRING[0]; (*Zeiger auf den Datenobjekt-Namen*)
		nDataObjMemType : {REDUND_UNREPLICABLE} USINT; (*Angabe über den Speicher-Typ des Datenobjekts*)
		nDataObjOption : {REDUND_UNREPLICABLE} UDINT; (*Angabe über die Option des Datenobjekts*)
	END_VAR
	VAR_OUTPUT
		nStatus : {REDUND_UNREPLICABLE} UINT; (*Fub-Status*)
		nDataObjIdent : {REDUND_UNREPLICABLE} UDINT; (*Ident des Datenobjekts*)
		pDataObjMem : {REDUND_UNREPLICABLE} UDINT; (*Zeiger auf die Daten des Datenobjekts*)
		nDataObjLen : {REDUND_UNREPLICABLE} UDINT; (*Länge des Datenobjekts (= Länge der Datei)*)
	END_VAR
	VAR
		eStep : {REDUND_UNREPLICABLE} DINT; (*Step-Nummer für die interne Schrittkette*)
		nStatusIntern : {REDUND_UNREPLICABLE} UINT; (*Interner Fub-Status*)
		fbDatObjInfo : {REDUND_UNREPLICABLE} DatObjInfo; (*Interner Fub*)
		fbDatObjDelete : {REDUND_UNREPLICABLE} DatObjDelete; (*Interner Fub*)
		fbFileOpen : {REDUND_UNREPLICABLE} FileOpen; (*Interner Fub*)
		fbDatObjCreate : {REDUND_UNREPLICABLE} DatObjCreate; (*Interner Fub*)
		fbFileRead : {REDUND_UNREPLICABLE} FileRead; (*Interner Fub*)
		fbFileClose : {REDUND_UNREPLICABLE} FileClose; (*Interner Fub*)
	END_VAR
END_FUNCTION_BLOCK

{REDUND_UNREPLICABLE} FUNCTION_BLOCK BrbSaveFileDataObj (*Speichert ein Datenobjekt in eine Datei*)
	VAR_INPUT
		pDevice : REFERENCE TO STRING[0]; (*Zeiger auf den Laufwerks-Namen*)
		pFile : REFERENCE TO STRING[0]; (*Zeiger auf den Datei-Namen*)
		pDataObjName : REFERENCE TO STRING[0]; (*Zeiger auf den Datenobjekt-Namen*)
	END_VAR
	VAR_OUTPUT
		nStatus : {REDUND_UNREPLICABLE} UINT; (*Fub-Status*)
	END_VAR
	VAR
		eStep : {REDUND_UNREPLICABLE} DINT; (*Step-Nummer für die interne Schrittkette*)
		nStatusIntern : {REDUND_UNREPLICABLE} UINT; (*Interner Fub-Status*)
		fbDatObjInfo : {REDUND_UNREPLICABLE} DatObjInfo; (*Interner Fub*)
		fbFileInfo : {REDUND_UNREPLICABLE} FileInfo; (*Interner Fub*)
		FileInfo : {REDUND_UNREPLICABLE} fiFILE_INFO; (*Interne Daten*)
		fbFileDelete : {REDUND_UNREPLICABLE} FileDelete; (*Interner Fub*)
		fbFileCreate : {REDUND_UNREPLICABLE} FileCreate; (*Interner Fub*)
		fbFileWrite : {REDUND_UNREPLICABLE} FileWrite; (*Interner Fub*)
		fbFileClose : {REDUND_UNREPLICABLE} FileClose; (*Interner Fub*)
	END_VAR
END_FUNCTION_BLOCK

{REDUND_UNREPLICABLE} FUNCTION_BLOCK BrbLoadFileBin (*Lädt eine Datei in eine Feld-Variable*) (*$GROUP=User,$CAT=User,$GROUPICON=User.png,$CATICON=User.png*)
	VAR_INPUT
		pDevice : REFERENCE TO STRING[0]; (*Zeiger auf den Laufwerks-Namen*)
		pFile : REFERENCE TO STRING[0]; (*Zeiger auf den Datei-Namen*)
		pVar : REFERENCE TO USINT; (*Zeiger auf die Feld-Variable*)
		nVarSize : {REDUND_UNREPLICABLE} UDINT; (*Größe der Feld-Variable*)
	END_VAR
	VAR_OUTPUT
		nStatus : {REDUND_UNREPLICABLE} UINT; (*Fub-Status*)
		nValidBytes : {REDUND_UNREPLICABLE} UDINT; (*Anzahl der gelesenen Bytes*)
	END_VAR
	VAR
		eStep : {REDUND_UNREPLICABLE} DINT; (*Step-Nummer für die interne Schrittkette*)
		nStatusIntern : {REDUND_UNREPLICABLE} UINT; (*Interner Fub-Status*)
		fbFileOpen : {REDUND_UNREPLICABLE} FileOpen; (*Interner Fub*)
		fbFileReadEx : {REDUND_UNREPLICABLE} FileReadEx; (*Interner Fub*)
		fbFileClose : {REDUND_UNREPLICABLE} FileClose; (*Interner Fub*)
	END_VAR
END_FUNCTION_BLOCK

FUNCTION BrbCheckFileName : UINT (*Ersetzt Sonderzeichen in einem Datei-Namen mit Unterstrichen*)
	VAR_INPUT
		pFileName : STRING[0]; (*Zeiger auf den Datei-Namen*)
	END_VAR
END_FUNCTION

FUNCTION BrbCheckFileEnding : BOOL (*Prüft die Endung eines Datei-Namens und berichtigt sie gegebenenfalls*)
	VAR_INPUT
		pFileName : STRING[0]; (*Zeiger auf den Datei-Namen*)
		pEnding : STRING[0]; (*Zeiger auf die Datei-Endung (mit oder ohne Punkt)*)
	END_VAR
END_FUNCTION

FUNCTION BrbCombinePath : UINT (*Fügt zwei Pfade oder einen Pfad und eine Datei-Namen zusammen*)
	VAR_INPUT
		pPath : STRING[0]; (*Zeiger auf Pfad*)
		pFilename : STRING[0]; (*Zeiger auf Pfad oder Datei-Namen*)
		pFilenameWithPath : STRING[0]; (*Zeiger auf den String, der das Ergebnis aufnimmt*)
	END_VAR
END_FUNCTION
(*Logger*)

{REDUND_UNREPLICABLE} FUNCTION_BLOCK BrbLoggerReadHierarchicalList (*Liest die zu einem definierten Logger-Eintrag gehörende Hierarchie-Liste von Einträgen aus*) (*$GROUP=User,$CAT=User,$GROUPICON=User.png,$CATICON=User.png*)
	VAR_INPUT
		sLogbookName : {REDUND_UNREPLICABLE} STRING[256]; (*Name des Logbuchs*)
		nStartRecordId : {REDUND_UNREPLICABLE} ArEventLogRecordIDType; (*RecordId, bei dem die Suche beginnen soll (0=Beginn bei jüngstem Eintrag)*)
		sObjectId : {REDUND_UNREPLICABLE} STRING[36]; (*ObjectId-Filter ('Entered by'-Angabe)*)
		nStartEventId : {REDUND_UNREPLICABLE} DINT; (*EventId oder ErrorNumber, bei dem die Liste beginnen soll (0=keine Filterung)*)
		eSeverities : {REDUND_UNREPLICABLE} BrbLogHierarchListSevFilter_ENUM; (*Bitweise codierte Filterung der Severities (0=keine Filterung)*)
		sLanguageCode : {REDUND_UNREPLICABLE} ArEventLogLanguageCodeType; (*Sprachkürzel*)
		nSearchEntryCountLimit : {REDUND_UNREPLICABLE} UDINT; (*Limitierung der durchsuchten Einträge (0=kein Limit)*)
		pLogList : {REDUND_UNREPLICABLE} UDINT; (*Zeiger auf die zu füllende Liste*)
		nLogListIndexMax : {REDUND_UNREPLICABLE} UINT; (*Maximaler Index der Liste*)
	END_VAR
	VAR_OUTPUT
		nListEntryCount : {REDUND_UNREPLICABLE} UINT; (*Anzahl der Einträge in der Liste*)
		nStatus : {REDUND_UNREPLICABLE} DINT; (*Fub-Status*)
	END_VAR
	VAR
		eStep : {REDUND_UNREPLICABLE} DINT; (*Step-Nummer für die interne Schrittkette*)
		sLastLogbookName : {REDUND_UNREPLICABLE} STRING[256]; (*Name des Logbuchs beim letzten Aufruf*)
		fbArEventLogGetIdent : {REDUND_UNREPLICABLE} ArEventLogGetIdent; (*Interner Fub*)
		nEventLogIdent : {REDUND_UNREPLICABLE} ArEventLogIdentType; (*Ident des Logbuchs*)
		ActEntry : {REDUND_UNREPLICABLE} BrbLogHierarchListEntry_TYP; (*Aktuell ermittelter Eintrag*)
		fbArEventLogGetLatestRecordID : {REDUND_UNREPLICABLE} ArEventLogGetLatestRecordID; (*Interner Fub*)
		fbArEventLogGetPreviousRecordID : {REDUND_UNREPLICABLE} ArEventLogGetPreviousRecordID; (*Interner Fub*)
		fbArEventLogRead : {REDUND_UNREPLICABLE} ArEventLogRead; (*Interner Fub*)
		fbArEventLogReadErrorNumber : {REDUND_UNREPLICABLE} ArEventLogReadErrorNumber; (*Interner Fub*)
		fbArEventLogReadObjectID : {REDUND_UNREPLICABLE} ArEventLogReadObjectID; (*Interner Fub*)
		fbArEventLogReadDescription : {REDUND_UNREPLICABLE} ArEventLogReadDescription; (*Interner Fub*)
		LogListManagement : {REDUND_UNREPLICABLE} BrbMemListManagement_Typ; (*Verwaltung der Liste*)
		nSearchEntryCount : {REDUND_UNREPLICABLE} UDINT; (*Anzahl der durchsuchten Einträge*)
		bFirstEntryIsListed : {REDUND_UNREPLICABLE} BOOL; (*Erster Eintrag lt. Filter eingetragen*)
	END_VAR
END_FUNCTION_BLOCK
(*TimeAndDate*)

FUNCTION BrbSetDtStruct : DATE_AND_TIME (*Setzt eine DTStructure-Zeit*) (*$GROUP=User,$CAT=User,$GROUPICON=User.png,$CATICON=User.png*)
	VAR_INPUT
		pDtStruct : DTStructure; (*Zeiger auf eine Zeit-Struktur*)
		nYear : UINT; (*Jahr*)
		nMonth : USINT; (*Monat*)
		nDay : USINT; (*Tage*)
		nHour : USINT; (*Stunde*)
		nMinute : USINT; (*Minute*)
		nSecond : USINT; (*Sekunde*)
		nMillisecond : UINT; (*Millisekunde*)
		nMicrosecond : UINT; (*Mikrosekunden*)
	END_VAR
END_FUNCTION

FUNCTION BrbSetDt : DATE_AND_TIME (*Setzt eine DATE_AND_TIME-Zeit*) (*$GROUP=User,$CAT=User,$GROUPICON=User.png,$CATICON=User.png*)
	VAR_INPUT
		nYear : UINT; (*Jahr*)
		nMonth : USINT; (*Monat*)
		nDay : USINT; (*Tage*)
		nHour : USINT; (*Stunde*)
		nMinute : USINT; (*Minute*)
		nSecond : USINT; (*Sekunde*)
	END_VAR
END_FUNCTION

FUNCTION BrbSetTimespan : TIME (*Setzt eine TIME-Zeitspanne*) (*$GROUP=User,$CAT=User,$GROUPICON=User.png,$CATICON=User.png*)
	VAR_INPUT
		nSign : SINT; (*Vorzeichen*)
		nDays : UDINT; (*Tage*)
		nHours : UDINT; (*Stunden*)
		nMinutes : UDINT; (*Minuten*)
		nSeconds : UDINT; (*Sekunden*)
		nMilliseconds : UDINT; (*Millisekunden*)
	END_VAR
END_FUNCTION

FUNCTION BrbSetTimespanT : TIME (*Setzt eine TIME-Zeitspanne*) (*$GROUP=User,$CAT=User,$GROUPICON=User.png,$CATICON=User.png*)
	VAR_INPUT
		pTimeText : STRING[0]; (*Zeiger auf die Text-Angabe*)
	END_VAR
END_FUNCTION

FUNCTION BrbGetTimeText : UINT (*Gibt die angegebene RTC-Zeit als Text zurück*)
	VAR_INPUT
		pTime : RTCtime_typ; (*Zeiger auf eine Zeit-Struktur*)
		pText : STRING[0]; (*Zeiger auf den String*)
		nTextSize : UDINT; (*Größe der String-Variablen*)
		pFormat : STRING[0]; (*Zeiger auf den Formatierungstext*)
	END_VAR
END_FUNCTION

FUNCTION BrbGetCurrentTimeText : UINT (*Gibt die aktuelle Zeit als Text zurück*)
	VAR_INPUT
		pText : STRING[0]; (*Zeiger auf den String*)
		nTextSize : UDINT; (*Größe der String-Variablen*)
		pFormat : STRING[0]; (*Zeiger auf den Formatierungstext*)
	END_VAR
END_FUNCTION

FUNCTION BrbGetTimeTextDtStruct : UINT (*Gibt die angegebene DtStruct-Zeit als Text zurück*)
	VAR_INPUT
		pTime : DTStructure; (*Zeiger auf eine Zeit-Struktur*)
		pText : STRING[0]; (*Zeiger auf den String*)
		nTextSize : UDINT; (*Größe der String-Variablen*)
		pFormat : STRING[0]; (*Zeiger auf den Formatierungstext*)
	END_VAR
END_FUNCTION

FUNCTION BrbGetTimeTextDt : UINT (*Gibt die angegebene DT-Zeit als Text zurück*)
	VAR_INPUT
		dtTime : DATE_AND_TIME; (*Zeiger auf eine DT-Zeit*)
		pText : STRING[0]; (*Zeiger auf den String*)
		nTextSize : UDINT; (*Größe der String-Variablen*)
		pFormat : STRING[0]; (*Zeiger auf den Formatierungstext*)
	END_VAR
END_FUNCTION

FUNCTION BrbGetDtFromTimeText : DATE_AND_TIME (*Wandelt einen Zeit-Text in eine Zeit um*)
	VAR_INPUT
		pTimeText : STRING[0]; (*Zeiger auf den Zeit-Text im Format*)
		pFormat : STRING[0]; (*Zeiger auf den Formatierungstext*)
	END_VAR
END_FUNCTION

FUNCTION BrbRtcTimeToDtStruct : UINT (*Wandelt eine RTC-Zeit in eine DtStruct-Zeit*)
	VAR_INPUT
		pRtcTime : RTCtime_typ; (*Zeiger auf eine Struktur "RTCtime_typ"*)
		pDtStruct : DTStructure; (*Zeiger auf eine Struktur "DTStructure"*)
	END_VAR
END_FUNCTION

FUNCTION BrbDtStructCompare : BOOL (*Vergleicht zwei DtStructures*)
	VAR_INPUT
		pDtStruct1 : DTStructure; (*Zeiger auf eine Struktur "DTStructure"*)
		eCompare : BrbTimeAndDateCompare_ENUM; (*Vergleichs-Angabe*)
		pDtStruct2 : DTStructure; (*Zeiger auf eine Struktur "DTStructure"*)
	END_VAR
END_FUNCTION

FUNCTION BrbDtStructAddDays : DATE_AND_TIME (*Addiert zu einer DTStructure die angegebenen Tage*)
	VAR_INPUT
		pDtStruct : DTStructure; (*Zeiger auf eine Struktur "DTStructure"*)
		nDays : DINT; (*Zu addierende Tage*)
	END_VAR
END_FUNCTION

FUNCTION BrbDtStructAddHours : DATE_AND_TIME (*Addiert zu einer DTStructure die angegebenen Stunden*)
	VAR_INPUT
		pDtStruct : DTStructure; (*Zeiger auf eine Struktur "DTStructure"*)
		nHours : DINT; (*Zu addierende Stunden*)
	END_VAR
END_FUNCTION

FUNCTION BrbDtStructAddMinutes : DATE_AND_TIME (*Addiert zu einer DTStructure die angegebenen Minuten*)
	VAR_INPUT
		pDtStruct : DTStructure; (*Zeiger auf eine Struktur "DTStructure"*)
		nMinutes : DINT; (*Zu addierende Minuten*)
	END_VAR
END_FUNCTION

FUNCTION BrbDtStructAddSeconds : DATE_AND_TIME (*Addiert zu einer DTStructure die angegebenen Sekunden*)
	VAR_INPUT
		pDtStruct : DTStructure; (*Zeiger auf eine Struktur "DTStructure"*)
		nSeconds : DINT; (*Zu addierende Sekunden*)
	END_VAR
END_FUNCTION

FUNCTION BrbDtStructAddMilliseconds : DATE_AND_TIME (*Addiert zu einer DTStructure die angegebenen Millisekunden*)
	VAR_INPUT
		pDtStruct : DTStructure; (*Zeiger auf eine Zeit-Struktur*)
		nMilliseconds : DINT; (*Millisekunden*)
	END_VAR
END_FUNCTION

FUNCTION BrbDtStructAddMillisecondsLReal : DATE_AND_TIME (*Addiert zu einer DTStructure die angegebenen Millisekunden*)
	VAR_INPUT
		pDtStruct : DTStructure; (*Zeiger auf eine Zeit-Struktur*)
		rMilliseconds : LREAL; (*Millisekunden*)
	END_VAR
END_FUNCTION

FUNCTION BrbGetTimeTextMs : UINT (*Gibt die angebenene Millisekunden-Zeit als Text zurück*) (*$GROUP=User*)
	VAR_INPUT
		nMilliseconds : DINT; (*Anzahl der Millisekunden*)
		pText : STRING[0]; (*Zeiger auf den String*)
		nTextSize : UDINT; (*Größe der String-Variablen*)
		pFormat : STRING[0]; (*Zeiger auf den Formatierungstext*)
		bClip : BOOL; (*Abziehen der nicht im Format berücksichtigten Teilwerte*)
	END_VAR
END_FUNCTION

FUNCTION BrbGetTimeDiffMsDtStruct : DINT (*Gibt die Zeit-Differenz zweier DtStruct-Zeiten in [ms] zurück*) (*$GROUP=User*)
	VAR_INPUT
		pTimeStampBase : DTStructure; (*Basis-Zeitstempel*)
		pTimeStampCompare : DTStructure; (*Vergleichs-Zeitstempel*)
	END_VAR
END_FUNCTION

FUNCTION BrbGetWeekdayDtStruct : BrbWeekdays_ENUM (*Ermittelt den Wochentag einer DTStructure*) (*$GROUP=User,$CAT=User,$GROUPICON=User.png,$CATICON=User.png*)
	VAR_INPUT
		pDtStruct : DTStructure; (*Zeiger auf eine Zeit-Struktur*)
	END_VAR
END_FUNCTION

FUNCTION BrbGetWeekdayDt : BrbWeekdays_ENUM (*Gibt den Wochentag einer DT-Zeit zurück*) (*$GROUP=User,$CAT=User,$GROUPICON=User.png,$CATICON=User.png*)
	VAR_INPUT
		dtTime : DATE_AND_TIME; (*Zeit-Angabe*)
	END_VAR
END_FUNCTION

{REDUND_UNREPLICABLE} FUNCTION_BLOCK BrbTimerSwitch (*Zeitschaltuhr für einen Kanal*)
	VAR_INPUT
		bEnable : {REDUND_UNREPLICABLE} BOOL; (*1=Baustein wird ausgeführt*)
		bCmdSwitchOff : {REDUND_UNREPLICABLE} BOOL; (*1=Ausgangs-Kanal wird ausgeschaltet*)
		bCmdSwitchOn : {REDUND_UNREPLICABLE} BOOL; (*1=Ausgangs-Kanal wird eingeschaltet*)
		bCmdToggle : {REDUND_UNREPLICABLE} BOOL; (*1=Ausgangs-Kanal wird umgeschaltet*)
		pUserTime : REFERENCE TO DTStructure; (*Optionaler Zeiger auf Benutzer-Zeitstempel*)
		Parameter : {REDUND_UNREPLICABLE} BrbTimerSwitchPar_TYP; (*Parameter-Struktur*)
	END_VAR
	VAR_OUTPUT
		bOut : {REDUND_UNREPLICABLE} BOOL; (*Ausgangs-Kanal*)
		dtsUsedTime : {REDUND_UNREPLICABLE} DTStructure; (*Verwendete Zeit*)
		nSwitchCount : {REDUND_UNREPLICABLE} UDINT; (*Anzahl der Schaltungen*)
	END_VAR
	VAR
		fbDTStructureGetTime : {REDUND_UNREPLICABLE} DTStructureGetTime; (*Interner Fub*)
		bLocked : {REDUND_UNREPLICABLE} BOOL; (*Interne Variable*)
		fbLock : {REDUND_UNREPLICABLE} TON; (*Interner Fub*)
		bClearOutOnNextCycle : {REDUND_UNREPLICABLE} BOOL; (*Interne Variable*)
	END_VAR
END_FUNCTION_BLOCK
(*Strings*)

FUNCTION BrbUsintToHex : UINT (*Wandelt einen Usint in einen Hex-String*)
	VAR_INPUT
		nValue : USINT; (*USINT-Wert*)
		pHex : STRING[0]; (*Zeiger auf den String*)
		nHexSize : UDINT; (*Größe der String-Variablen*)
		bWithPraefix : BOOL; (*1=Mit Präfix '0x'*)
	END_VAR
END_FUNCTION

FUNCTION BrbUsintArrayToHex : UINT (*Wandelt ein Usint-Array in einen Hex-String*) (*$GROUP=User,$CAT=User,$GROUPICON=User.png,$CATICON=User.png*)
	VAR_INPUT
		pArray : REFERENCE TO USINT; (*Zeiger auf das Array*)
		nArrayLength : DINT; (*Länge des Arrays*)
		pHex : STRING[0]; (*Zeiger auf den String*)
		nHexSize : UDINT; (*Größe der String-Variablen*)
		bDescending : BOOL; (*0=Aufsteigend, 1=Absteigend*)
	END_VAR
END_FUNCTION

FUNCTION BrbHexToUsintArray : UINT (*Wandelt einen Hex-String in ein Usint-Array*) (*$GROUP=User,$CAT=User,$GROUPICON=User.png,$CATICON=User.png*)
	VAR_INPUT
		pHex : STRING[0]; (*Zeiger auf den String*)
		pArray : REFERENCE TO USINT; (*Zeiger auf das Array*)
		nArrayLength : DINT; (*Länge des Arrays*)
		bDescending : BOOL; (*0=Aufsteigend, 1=Absteigend*)
	END_VAR
END_FUNCTION

FUNCTION BrbUdintToAscii : UINT (*Wandelt einen UDINT-Wert zu einem String*)
	VAR_INPUT
		nValue : UDINT; (*UDINT-Wert*)
		pText : STRING[0]; (*Zeiger auf den String*)
	END_VAR
END_FUNCTION

FUNCTION BrbAsciiToUdint : UDINT (*Wandelt einen String zu einem UDINT-Wert*)
	VAR_INPUT
		pText : STRING[0]; (*Zeiger auf den String*)
	END_VAR
END_FUNCTION

FUNCTION BrbUdintToHex : UINT (*Wandelt einen Udint in einen Hex-String*)
	VAR_INPUT
		nValue : UDINT; (*UDINT-Wert*)
		pHex : STRING[0]; (*Zeiger auf den String*)
		nHexSize : UDINT; (*Größe der String-Variablen*)
		bWithPraefix : BOOL; (*1=Mit Präfix '0x'*)
	END_VAR
END_FUNCTION

FUNCTION BrbHexToUdint : UDINT (*Wandelt einen Hex-String in einen Udint*)
	VAR_INPUT
		pHex : STRING[0]; (*Zeiger auf den String*)
	END_VAR
END_FUNCTION

FUNCTION BrbUdintToBin : UINT (*Wandelt einen Udint-Wert in einen Binär-String*) (*$GROUP=User,$CAT=User,$GROUPICON=User.png,$CATICON=User.png*)
	VAR_INPUT
		nValue : UDINT; (*UDINT-Wert*)
		pBin : STRING[0]; (*Zeiger auf den String*)
		nBinSize : UDINT; (*Größe der String-Variablen*)
		bWithPraefix : BOOL; (*1=Mit Präfix '%'*)
	END_VAR
END_FUNCTION

FUNCTION BrbDintToHex : UINT (*Wandelt einen DINT in einen Hex-String*) (*$GROUP=User*)
	VAR_INPUT
		nValue : DINT; (*DINT-Wert*)
		pHex : STRING[0]; (*Zeiger auf den String*)
		nHexSize : UDINT; (*Größe der String-Variablen*)
		bWithPraefix : BOOL; (*1=Mit Präfix '0x'*)
	END_VAR
END_FUNCTION

FUNCTION BrbHexToDint : DINT (*Wandelt einen Hex-String in einen Dint*) (*$GROUP=User*)
	VAR_INPUT
		pHex : STRING[0]; (*Zeiger auf den String*)
	END_VAR
END_FUNCTION

FUNCTION BrbAsciiFieldToString : BOOL (*Wandelt ein Ascii-Feld in einen lesbaren Text*)
	VAR_INPUT
		pAsciiField : REFERENCE TO USINT; (*Zeiger auf das Ascii-Feld*)
		nAsciiFieldLen : UDINT; (*Länge des Ascii-Felds*)
		nFinalAsciiCharCount : UDINT; (*Anzahl der letzten Ascii-Zeichen, die auf jeden Fall enthalten sein sollten*)
		pText : STRING[0]; (*Zeiger auf den String*)
		nTextSize : UDINT; (*Größe der String-Variablen*)
	END_VAR
END_FUNCTION

FUNCTION BrbStringGetIndexOf : DINT (*Gibt den ersten Index eines zu suchenden Textes zurück*)
	VAR_INPUT
		pText : STRING[0]; (*Zeiger auf den ganzen Text*)
		pFind : STRING[0]; (*Zeiger auf den zu suchenden Text*)
		nTextLen : UDINT; (*Länge des ganzen Textes*)
	END_VAR
END_FUNCTION

FUNCTION BrbStringGetLastIndexOf : DINT (*Gibt den letzten Index eines zu suchenden Textes zurück*)
	VAR_INPUT
		pText : STRING[0]; (*Zeiger auf den ganzen Text*)
		pFind : STRING[0]; (*Zeiger auf den zu suchenden Text*)
		nTextLen : UDINT; (*Länge des ganzen Textes*)
	END_VAR
END_FUNCTION

FUNCTION BrbStringGetAdrOf : STRING[0] (*Gibt die erste Adresse eines zu suchenden Textes zurück*)
	VAR_INPUT
		pText : STRING[0]; (*Zeiger auf den ganzen Text*)
		pFind : STRING[0]; (*Zeiger auf den zu suchenden Text*)
		nTextLen : UDINT; (*Länge des ganzen Textes*)
	END_VAR
END_FUNCTION

FUNCTION BrbStringGetLastAdrOf : STRING[0] (*Gibt die letzte Adresse eines zu suchenden Textes zurück*)
	VAR_INPUT
		pText : STRING[0]; (*Zeiger auf den ganzen Text*)
		pFind : STRING[0]; (*Zeiger auf den zu suchenden Text*)
		nTextLen : UDINT; (*Länge des ganzen Textes*)
	END_VAR
END_FUNCTION

FUNCTION BrbStringStartsWith : BOOL (*Gibt zurück, ob ein Text mit einer bestimmten Zeichenfolge beginnt*)
	VAR_INPUT
		pText : STRING[0]; (*Zeiger auf den ganzen Text*)
		pFind : STRING[0]; (*Zeiger auf den zu suchenden Text*)
	END_VAR
END_FUNCTION

FUNCTION BrbStringEndsWith : BOOL (*Gibt zurück, ob ein Text mit einer bestimmten Zeichenfolge endet*)
	VAR_INPUT
		pText : STRING[0]; (*Zeiger auf den ganzen Text*)
		pFind : STRING[0]; (*Zeiger auf den zu suchenden Text*)
	END_VAR
END_FUNCTION

FUNCTION BrbStringGetSubText : STRING[0] (*Gibt eine Zeichenfolge innerhalb eines Textes zurück*)
	VAR_INPUT
		pText : STRING[0]; (*Zeiger auf den ganzen Text*)
		nIndex : UDINT; (*Start-Index*)
		nLen : UDINT; (*Länge*)
		pSubText : STRING[0]; (*Zeiger auf eine String-Variable, die das Ergebnis aufnimmt*)
	END_VAR
END_FUNCTION

FUNCTION BrbStringGetSubTextByLen : STRING[0] (*Gibt eine Zeichenfolge innerhalb eines Textes zurück*)
	VAR_INPUT
		pStart : STRING[0]; (*Zeiger auf den Start der Zeichenfolge*)
		nLen : UDINT; (*Länge*)
		pSubText : STRING[0]; (*Zeiger auf eine String-Variable, die das Ergebnis aufnimmt*)
	END_VAR
END_FUNCTION

FUNCTION BrbStringGetSubTextByAdr : STRING[0] (*Gibt eine Zeichenfolge innerhalb eines Textes zurück*)
	VAR_INPUT
		pStart : STRING[0]; (*Zeiger auf den Start der Zeichenfolge*)
		pEnd : STRING[0]; (*Zeiger auf das Ende der Zeichenfolge*)
		pSubText : STRING[0]; (*Zeiger auf eine String-Variable, die das Ergebnis aufnimmt*)
	END_VAR
END_FUNCTION

FUNCTION BrbStringAppend : UDINT (*Hängt eine Zeichenfolge an einen Text (Ersatz für strcat)*)
	VAR_INPUT
		pText : STRING[0]; (*Zeiger auf den ganzen Text*)
		pTextAppend : STRING[0]; (*Zeiger auf den anzuhängenden Text*)
		pTextOffset : REFERENCE TO UDINT; (*Zeiger auf das momentane Ende*)
	END_VAR
END_FUNCTION

FUNCTION BrbStringCut : STRING[0] (*Schneidet eine Zeichenfolge aus einem Text heraus*)
	VAR_INPUT
		pText : STRING[0]; (*Zeiger auf den ganzen Text*)
		nCutIndex : UDINT; (*Start-Index der Schneidung*)
		nCutLen : UDINT; (*Länge der Schneidung*)
		pCut : STRING[0]; (*Zeiger auf eine String-Variable, die die herausgeschnittene Zeichenfolge aufnimmt*)
	END_VAR
END_FUNCTION

FUNCTION BrbStringCutFromLastSeparator : UDINT (*Schneidet die Zeichenfolge ab dem letzten Trennzeichen in einem Text ab*)
	VAR_INPUT
		pText : STRING[0]; (*Zeiger auf den ganzen Text*)
		pSeparator : STRING[0]; (*Zeiger auf den zu suchenden Text*)
		pCut : STRING[0]; (*Zeiger auf eine String-Variable, die die herausgeschnittene Zeichenfolge aufnimmt*)
	END_VAR
END_FUNCTION

FUNCTION BrbStringInsert : STRING[0] (*Fügt eine Zeichenfolge in einen Text ein*)
	VAR_INPUT
		pText : STRING[0]; (*Zeiger auf den ganzen Text*)
		nInsertIndex : UDINT; (*Start-Index der Einfügung*)
		pInsert : STRING[0]; (*Zeiger auf die einzufügende Zeichenfolge*)
	END_VAR
END_FUNCTION

FUNCTION BrbStringReplace : UDINT (*Ersetzt eine Zeichenfolge in einem Text durch eine andere*)
	VAR_INPUT
		pText : STRING[0]; (*Zeiger auf den ganzen Text*)
		pFind : STRING[0]; (*Zeiger auf die zu ersetzende Zeichenfolge*)
		pReplace : STRING[0]; (*Zeiger auf die ersetzende Zeichenfolge*)
	END_VAR
END_FUNCTION

FUNCTION BrbStringPadLeft : BOOL (*Füllt einen String auf der linken Seite mit einem Füllzeichen auf eine bestimme Länge*)
	VAR_INPUT
		pText : STRING[0]; (*Zeiger auf den Text*)
		pFillChar : STRING[0]; (*Zeiger auf das Füllzeichen*)
		nLen : UDINT; (*Länge, auf die gefüllt werden soll*)
	END_VAR
END_FUNCTION

FUNCTION BrbStringPadRight : BOOL (*Füllt einen String auf der rechten Seite mit einem Füllzeichen auf eine bestimme Länge*)
	VAR_INPUT
		pText : STRING[0]; (*Zeiger auf den Text*)
		pFillChar : STRING[0]; (*Zeiger auf das Füllzeichen*)
		nLen : UDINT; (*Länge, auf die gefüllt werden soll*)
	END_VAR
END_FUNCTION

FUNCTION BrbStringTrimLeft : BOOL (*Schneidet eine Zeichenfolge auf der linken Seite eines Textes heraus*)
	VAR_INPUT
		pText : STRING[0]; (*Zeiger auf den Text*)
		pTrim : STRING[0]; (*Zeiger auf die herauszuschneidene Zeichenfolge*)
	END_VAR
END_FUNCTION

FUNCTION BrbStringTrimRight : BOOL (*Schneidet eine Zeichenfolge auf der rechten Seite eines Textes heraus*)
	VAR_INPUT
		pText : STRING[0]; (*Zeiger auf den Text*)
		pTrim : STRING[0]; (*Zeiger auf die herauszuschneidene Zeichenfolge*)
	END_VAR
END_FUNCTION

FUNCTION BrbStringSplit : UDINT (*Spaltet einen Text in mehrere Strings aufgrund eines Trennzeichens*)
	VAR_INPUT
		pText : STRING[0]; (*Zeiger auf den Text*)
		pSep : STRING[0]; (*Zeiger auf das Trennzeichen*)
		pSplitArray : UDINT; (*Zeiger auf ein String-Array*)
		nArrayIndexMax : UDINT; (*Maximaler Index des String-Arrays*)
		nEntrySize : UDINT; (*Größe eines Strings im String-Array*)
	END_VAR
END_FUNCTION

FUNCTION BrbStringSplitEmpty : UDINT (*Spaltet einen Text in mehrere Strings aufgrund eines Trennzeichens (inkl. Leer-Strings)*) (*$GROUP=User,$CAT=User,$GROUPICON=User.png,$CATICON=User.png*)
	VAR_INPUT
		pText : STRING[0]; (*Zeiger auf den Text*)
		pSep : STRING[0]; (*Zeiger auf das Trennzeichen*)
		pSplitArray : UDINT; (*Zeiger auf ein String-Array*)
		nArrayIndexMax : UDINT; (*Maximaler Index des String-Arrays*)
		nEntrySize : UDINT; (*Maximaler Index des String-Arrays*)
	END_VAR
END_FUNCTION

FUNCTION BrbStringConvertRealFromExp : UINT (*Konvertiert eine exponentielle Notation in einen Real-Wert*)
	VAR_INPUT
		pValue : STRING[0]; (*Zeiger auf den Wert-Text*)
		pResult : STRING[0]; (*Zeiger auf eine String-Variable, die das Ergebnis aufnimmt*)
		nResultSize : UDINT; (*Größe der Ergebnis-Variable*)
	END_VAR
END_FUNCTION

FUNCTION BrbStringConvertRealToExp : UINT (*Konvertiert einen Real-Wert in eine exponentielle Notation*)
	VAR_INPUT
		pValue : STRING[0]; (*Zeiger auf den Wert-Text*)
		pResult : STRING[0]; (*Zeiger auf eine String-Variable, die das Ergebnis aufnimmt*)
		nResultSize : UDINT; (*Größe der Ergebnis-Variable*)
	END_VAR
END_FUNCTION

FUNCTION BrbStringFormatFractionDigits : UINT (*Formatiert einen Real-String-Wert auf Nachkommastellen*)
	VAR_INPUT
		pValue : STRING[0]; (*Zeiger auf den Wert-Text*)
		nValueSize : UDINT; (*Größe der Variable*)
		nFractionsDigits : UINT; (*Anzahl der Nachkomma-Stellen*)
	END_VAR
END_FUNCTION

FUNCTION BrbStringSwap : BOOL (*Dreht die Reihenfolge der Zeichen in einem Text*)
	VAR_INPUT
		pText : STRING[0]; (*Zeiger auf den zu drehenden Text*)
		pSwapped : STRING[0]; (*Zeiger auf eine String-Variable, die das Ergebnis aufnimmt*)
		nSwappedSize : UDINT; (*Größe der String-Variablen*)
	END_VAR
END_FUNCTION

FUNCTION BrbStringToUpper : BOOL (*Konvertiert einen String zu Großbuchstaben*)
	VAR_INPUT
		pText : STRING[0]; (*Zeiger auf den Text*)
	END_VAR
END_FUNCTION

FUNCTION BrbStringToLower : BOOL (*Konvertiert einen String zu Kleinbuchstaben*)
	VAR_INPUT
		pText : STRING[0]; (*Zeiger auf den Text*)
	END_VAR
END_FUNCTION

FUNCTION BrbStringIsNumerical : BOOL (*Gibt zurück, ob ein Text eine Nummer enthält*)
	VAR_INPUT
		pText : STRING[0]; (*Zeiger auf den Text*)
	END_VAR
END_FUNCTION

FUNCTION BrbStringIsHex : BOOL (*Gibt zurück, ob ein Text eine hexadezimale Nummer enthält*) (*$GROUP=User*)
	VAR_INPUT
		pText : STRING[0]; (*Zeiger auf den Text*)
		bLowCaseAllowed : BOOL; (*1=Kleinbuchstaben (a..f) sind erlaubt*)
	END_VAR
END_FUNCTION

FUNCTION BrbStringCountText : UDINT (*Zählt das Vorkommen einer Zeichenfolge innerhalb eines Texts*) (*$GROUP=User*)
	VAR_INPUT
		pText : STRING[0]; (*Zeiger auf den ganzen Text*)
		pFind : STRING[0]; (*Zeiger auf den zu suchenden Text*)
		nTextLen : UDINT; (*Länge des ganzen Textes*)
	END_VAR
END_FUNCTION

FUNCTION BrbStringRepeat : UDINT (*Wiederholt eine Zeichenfolge bis zu einer angegebenen Zeichenanzahl*) (*$GROUP=User,$CAT=User,$GROUPICON=User.png,$CATICON=User.png*)
	VAR_INPUT
		pText : STRING[0]; (*Zeiger auf den ganzen Text*)
		nTextSize : UDINT; (*Größe des Text-Strings*)
		pRepeat : STRING[0]; (*Zeiger auf die zu wiederholende Zeichenfolge*)
		nLen : UDINT; (*Anzahl der Zeichen, bei dem die Wiederholungen enden*)
	END_VAR
END_FUNCTION

FUNCTION BrbStringCopy : UDINT (*Sicheres Kopieren eines Strings*) (*$GROUP=User,$CAT=User,$GROUPICON=User.png,$CATICON=User.png*)
	VAR_INPUT
		pDest : STRING[0]; (*Zeiger auf den Zielstring*)
		pSrc : STRING[0]; (*Zeiger auf den Quellstring*)
		nDestSize : UDINT; (*Größe des Zielstrings*)
	END_VAR
END_FUNCTION

FUNCTION BrbStringCat : UDINT (*Sicheres Anhängen an einen String*) (*$GROUP=User,$CAT=User,$GROUPICON=User.png,$CATICON=User.png*)
	VAR_INPUT
		pDest : STRING[0]; (*Zeiger auf den Zielstring*)
		pSrc : STRING[0]; (*Zeiger auf den Quellstring*)
		nDestSize : UDINT; (*Größe des Zielstrings*)
	END_VAR
END_FUNCTION
(*WcStrings*)

FUNCTION BrbWcCopyStringToWString : UINT (*Kopiert einen STRING auf einen WSTRING*) (*$GROUP=User*)
	VAR_INPUT
		pWcString : WSTRING[0]; (*Zeiger auf WSTRING*)
		pString : STRING[0]; (*Zeiger auf STRING*)
	END_VAR
END_FUNCTION

FUNCTION BrbWcCopyWStringToString : UINT (*Kopiert einen WSTRING auf einen STRING*) (*$GROUP=User*)
	VAR_INPUT
		pString : STRING[0]; (*Zeiger auf STRING*)
		pWcString : WSTRING[0]; (*Zeiger auf WSTRING*)
	END_VAR
END_FUNCTION

FUNCTION BrbWcStringGetIndexOf : DINT (*Gibt den ersten Index eines zu suchenden Textes zurück*) (*$GROUP=User*)
	VAR_INPUT
		pText : WSTRING[0]; (*Zeiger auf den ganzen Text*)
		pFind : WSTRING[0]; (*Zeiger auf den zu suchenden Text*)
		nTextLen : UDINT; (*Länge des ganzen Textes*)
	END_VAR
END_FUNCTION

FUNCTION BrbWcStringGetLastIndexOf : DINT (*Gibt den letzten Index eines zu suchenden Textes zurück*) (*$GROUP=User*)
	VAR_INPUT
		pText : WSTRING[0]; (*Zeiger auf den ganzen Text*)
		pFind : WSTRING[0]; (*Zeiger auf den zu suchenden Text*)
		nTextLen : UDINT; (*Länge des ganzen Textes*)
	END_VAR
END_FUNCTION

FUNCTION BrbWcStringGetAdrOf : UDINT (*Gibt die erste Adresse eines zu suchenden Textes zurück*) (*$GROUP=User*)
	VAR_INPUT
		pText : WSTRING[0]; (*Zeiger auf den ganzen Text*)
		pFind : WSTRING[0]; (*Zeiger auf den zu suchenden Text*)
		nTextLen : UDINT; (*Länge des ganzen Textes*)
	END_VAR
END_FUNCTION

FUNCTION BrbWcStringGetLastAdrOf : UDINT (*Gibt die letzte Adresse eines zu suchenden Textes zurück*) (*$GROUP=User*)
	VAR_INPUT
		pText : WSTRING[0]; (*Zeiger auf den ganzen Text*)
		pFind : WSTRING[0]; (*Zeiger auf den zu suchenden Text*)
		nTextLen : UDINT; (*Länge des ganzen Textes*)
	END_VAR
END_FUNCTION

FUNCTION BrbWcStringStartsWith : BOOL (*Gibt zurück, ob ein Text mit einer bestimmten Zeichenfolge beginnt*) (*$GROUP=User*)
	VAR_INPUT
		pText : WSTRING[0]; (*Zeiger auf den ganzen Text*)
		pFind : WSTRING[0]; (*Zeiger auf den zu suchenden Text*)
	END_VAR
END_FUNCTION

FUNCTION BrbWcStringEndsWith : BOOL (*Gibt zurück, ob ein Text mit einer bestimmten Zeichenfolge endet*) (*$GROUP=User*)
	VAR_INPUT
		pText : WSTRING[0]; (*Zeiger auf den ganzen Text*)
		pFind : WSTRING[0]; (*Zeiger auf den zu suchenden Text*)
	END_VAR
END_FUNCTION

FUNCTION BrbWcStringGetSubText : UDINT (*Gibt eine Zeichenfolge innerhalb eines Textes zurück*) (*$GROUP=User*)
	VAR_INPUT
		pText : WSTRING[0]; (*Zeiger auf den ganzen Text*)
		nIndex : UDINT; (*Start-Index*)
		nLen : UDINT; (*Länge*)
		pSubText : WSTRING[0]; (*Zeiger auf eine WcString-Variable, die das Ergebnis aufnimmt*)
	END_VAR
END_FUNCTION

FUNCTION BrbWcStringGetSubTextByLen : UDINT (*Gibt eine Zeichenfolge innerhalb eines Textes zurück*) (*$GROUP=User*)
	VAR_INPUT
		pStart : WSTRING[0]; (*Zeiger auf den Start der Zeichenfolge*)
		nLen : UDINT; (*Länge*)
		pSubText : WSTRING[0]; (*Zeiger auf eine WcString-Variable, die das Ergebnis aufnimmt*)
	END_VAR
END_FUNCTION

FUNCTION BrbWcStringGetSubTextByAdr : UDINT (*Gibt eine Zeichenfolge innerhalb eines Textes zurück*) (*$GROUP=User*)
	VAR_INPUT
		pStart : WSTRING[0]; (*Zeiger auf den Start der Zeichenfolge*)
		pEnd : WSTRING[0]; (*Zeiger auf das Ende der Zeichenfolge*)
		pSubText : WSTRING[0]; (*Zeiger auf eine WcString-Variable, die das Ergebnis aufnimmt*)
	END_VAR
END_FUNCTION

FUNCTION BrbWcStringAppend : UDINT (*Hängt eine Zeichenfolge an einen Text (Ersatz für brwcscat)*) (*$GROUP=User*)
	VAR_INPUT
		pText : WSTRING[0]; (*Zeiger auf den ganzen Text*)
		pTextAppend : WSTRING[0]; (*Zeiger auf den anzuhängenden Text*)
		pTextOffset : REFERENCE TO UDINT; (*Zeiger auf das momentane Ende*)
	END_VAR
END_FUNCTION

FUNCTION BrbWcStringCut : UDINT (*Schneidet eine Zeichenfolge aus einem Text heraus*) (*$GROUP=User*)
	VAR_INPUT
		pText : WSTRING[0]; (*Zeiger auf den ganzen Text*)
		nCutIndex : UDINT; (*Start-Index der Schneidung*)
		nCutLen : UDINT; (*Länge der Schneidung*)
		pCut : WSTRING[0]; (*Zeiger auf eine WcString-Variable, die die herausgeschnittene Zeichenfolge aufnimmt*)
	END_VAR
END_FUNCTION

FUNCTION BrbWcStringInsert : UDINT (*Fügt eine Zeichenfolge in einen Text ein*) (*$GROUP=User*)
	VAR_INPUT
		pText : WSTRING[0]; (*Zeiger auf den ganzen Text*)
		nInsertIndex : UDINT; (*Start-Index der Einfügung*)
		pInsert : WSTRING[0]; (*Zeiger auf die einzufügende Zeichenfolge*)
	END_VAR
END_FUNCTION

FUNCTION BrbWcStringReplace : UDINT (*Ersetzt eine Zeichenfolge in einem Text durch eine andere*) (*$GROUP=User*)
	VAR_INPUT
		pText : WSTRING[0]; (*Zeiger auf den ganzen Text*)
		pFind : WSTRING[0]; (*Zeiger auf die zu ersetzende Zeichenfolge*)
		pReplace : WSTRING[0]; (*Zeiger auf die ersetzende Zeichenfolge*)
	END_VAR
END_FUNCTION

FUNCTION BrbWcStringPadLeft : BOOL (*Füllt einen String auf der linken Seite mit einem Füllzeichen auf eine bestimme Länge*) (*$GROUP=User*)
	VAR_INPUT
		pText : WSTRING[0]; (*Zeiger auf den Text*)
		pFillChar : WSTRING[0]; (*Zeiger auf das Füllzeichen*)
		nLen : UDINT; (*Länge, auf die gefüllt werden soll*)
	END_VAR
END_FUNCTION

FUNCTION BrbWcStringPadRight : BOOL (*Füllt einen String auf der rechten Seite mit einem Füllzeichen auf eine bestimme Länge*) (*$GROUP=User*)
	VAR_INPUT
		pText : WSTRING[0]; (*Zeiger auf den Text*)
		pFillChar : WSTRING[0]; (*Zeiger auf das Füllzeichen*)
		nLen : UDINT; (*Länge, auf die gefüllt werden soll*)
	END_VAR
END_FUNCTION

FUNCTION BrbWcStringTrimLeft : BOOL (*Schneidet eine Zeichenfolge auf der linken Seite eines Textes heraus*) (*$GROUP=User*)
	VAR_INPUT
		pText : WSTRING[0]; (*Zeiger auf den Text*)
		pTrim : WSTRING[0]; (*Zeiger auf die herauszuschneidene Zeichenfolge*)
	END_VAR
END_FUNCTION

FUNCTION BrbWcStringTrimRight : BOOL (*Schneidet eine Zeichenfolge auf der rechten Seite eines Textes heraus*) (*$GROUP=User*)
	VAR_INPUT
		pText : WSTRING[0]; (*Zeiger auf den Text*)
		pTrim : WSTRING[0]; (*Zeiger auf die herauszuschneidene Zeichenfolge*)
	END_VAR
END_FUNCTION

FUNCTION BrbWcStringToUpper : BOOL (*Konvertiert einen WcString zu Großbuchstaben*) (*$GROUP=User*)
	VAR_INPUT
		pText : WSTRING[0]; (*Zeiger auf den Text*)
	END_VAR
END_FUNCTION

FUNCTION BrbWcStringToLower : BOOL (*Konvertiert einen WcString zu Kleinbuchstaben*) (*$GROUP=User*)
	VAR_INPUT
		pText : WSTRING[0]; (*Zeiger auf den Text*)
	END_VAR
END_FUNCTION

FUNCTION BrbWcStringIsNumerical : BOOL (*Gibt zurück, ob ein Text eine Nummer enthält*) (*$GROUP=User*)
	VAR_INPUT
		pText : WSTRING[0]; (*Zeiger auf den Text*)
	END_VAR
END_FUNCTION

FUNCTION BrbWcStringIsHex : BOOL (*Gibt zurück, ob ein Text eine hexadezimale Nummer enthält*) (*$GROUP=User*)
	VAR_INPUT
		pText : WSTRING[80]; (*Zeiger auf den Text*)
		bLowCaseAllowed : BOOL; (*1=Kleinbuchstaben (a..f) sind erlaubt*)
	END_VAR
END_FUNCTION

FUNCTION BrbWcStringCountText : UDINT (*Zählt das Vorkommen einer Zeichenfolge innerhalb eines Texts*) (*$GROUP=User*)
	VAR_INPUT
		pText : WSTRING[0]; (*Zeiger auf den ganzen Text*)
		pFind : WSTRING[0]; (*Zeiger auf den zu suchenden Text*)
		nTextLen : UDINT; (*Länge des ganzen Textes*)
	END_VAR
END_FUNCTION

FUNCTION BrbWcStringRepeat : UDINT (*Wiederholt eine Zeichenfolge bis zu einer angegebenen Zeichenanzahl*) (*$GROUP=User,$CAT=User,$GROUPICON=User.png,$CATICON=User.png*)
	VAR_INPUT
		pText : WSTRING[0]; (*Zeiger auf den ganzen Text*)
		nTextSize : UDINT; (*Größe des Text-Strings*)
		pRepeat : WSTRING[0]; (*Zeiger auf die zu wiederholende Zeichenfolge*)
		nLen : UDINT; (*Anzahl der Zeichen, bei dem die Wiederholungen enden*)
	END_VAR
END_FUNCTION
(*BigDataTypes*)
(*BigDataTypes - Uint64*)

FUNCTION BrbUint64FromString : DINT (*Wandelt einen String in eine Uint64-Wert*) (*$GROUP=User,$CAT=User,$GROUPICON=User.png,$CATICON=User.png*)
	VAR_INPUT
		pUint64 : BrbUint64_TYP; (*Zeiger auf die Uint64-Struktur*)
		pText : STRING[0]; (*Zeiger auf den String*)
	END_VAR
END_FUNCTION

FUNCTION BrbUint64ToString : DINT (*Wandelt einen Uint64-Wert zu einem String*) (*$GROUP=User,$CAT=User,$GROUPICON=User.png,$CATICON=User.png*)
	VAR_INPUT
		pUint64 : BrbUint64_TYP; (*Zeiger auf die Uint64-Struktur*)
		pText : STRING[0]; (*Zeiger auf den String*)
		nTextSize : UDINT; (*Größe des Text-Strings*)
	END_VAR
END_FUNCTION

FUNCTION BrbUint64Compare : SINT (*Vergleicht zwei Uint64 auf kleiner, größer oder gleich*) (*$GROUP=User,$CAT=User,$GROUPICON=User.png,$CATICON=User.png*)
	VAR_INPUT
		pOperand0 : BrbUint64_TYP; (*Zeiger auf die erste Uint64-Struktur*)
		pOperand1 : BrbUint64_TYP; (*Zeiger auf die zweite Uint64-Struktur*)
	END_VAR
END_FUNCTION

FUNCTION BrbUint64Inc : DINT (*Inkrementiert einen Uint64-Wert um 1*) (*$GROUP=User,$CAT=User,$GROUPICON=User.png,$CATICON=User.png*)
	VAR_INPUT
		pUint64 : BrbUint64_TYP; (*Zeiger auf die Uint64-Struktur*)
	END_VAR
END_FUNCTION

FUNCTION BrbUint64Dec : DINT (*Dekrementiert einen Uint64-Wert um 1*) (*$GROUP=User,$CAT=User,$GROUPICON=User.png,$CATICON=User.png*)
	VAR_INPUT
		pUint64 : BrbUint64_TYP; (*Zeiger auf die Uint64-Struktur*)
	END_VAR
END_FUNCTION

FUNCTION BrbUint64Calculate : DINT (*Rechnet mit zwei Uint64*) (*$GROUP=User,$CAT=User,$GROUPICON=User.png,$CATICON=User.png*)
	VAR_INPUT
		pOperand0 : BrbUint64_TYP; (*Zeiger auf die erste Uint64-Struktur*)
		pOperand1 : BrbUint64_TYP; (*Zeiger auf die zweite Uint64-Struktur*)
		eOperator : BrbDt64Operator_ENUM; (*Operator-Angabe (Add, Subtract, Multiply, Divide)*)
	END_VAR
END_FUNCTION
(*BigDataTypes - Int64*)

FUNCTION BrbInt64FromString : DINT (*Wandelt einen String in eine Int64-Wert*) (*$GROUP=User,$CAT=User,$GROUPICON=User.png,$CATICON=User.png*)
	VAR_INPUT
		pInt64 : BrbInt64_TYP; (*Zeiger auf die Int64-Struktur*)
		pText : STRING[0]; (*Zeiger auf den String*)
	END_VAR
END_FUNCTION

FUNCTION BrbInt64ToString : DINT (*Wandelt einen Int64-Wert zu einem String*) (*$GROUP=User,$CAT=User,$GROUPICON=User.png,$CATICON=User.png*)
	VAR_INPUT
		pInt64 : BrbInt64_TYP; (*Zeiger auf die Int64-Struktur*)
		pText : STRING[0]; (*Zeiger auf den String*)
		nTextSize : UDINT; (*Größe des Text-Strings*)
	END_VAR
END_FUNCTION

FUNCTION BrbInt64Compare : SINT (*Vergleicht zwei Int64 auf kleiner, größer oder gleich*) (*$GROUP=User,$CAT=User,$GROUPICON=User.png,$CATICON=User.png*)
	VAR_INPUT
		pOperand0 : BrbInt64_TYP; (*Zeiger auf die erste Int64-Struktur*)
		pOperand1 : BrbInt64_TYP; (*Zeiger auf die zweite Int64-Struktur*)
	END_VAR
END_FUNCTION

FUNCTION BrbInt64Inc : DINT (*Inkrementiert einen Int64-Wert um 1*) (*$GROUP=User,$CAT=User,$GROUPICON=User.png,$CATICON=User.png*)
	VAR_INPUT
		pInt64 : BrbInt64_TYP; (*Zeiger auf die Int64-Struktur*)
	END_VAR
END_FUNCTION

FUNCTION BrbInt64Dec : DINT (*Dekrementiert einen Int64-Wert um 1*) (*$GROUP=User,$CAT=User,$GROUPICON=User.png,$CATICON=User.png*)
	VAR_INPUT
		pInt64 : BrbInt64_TYP; (*Zeiger auf die Int64-Struktur*)
	END_VAR
END_FUNCTION

FUNCTION BrbInt64Calculate : DINT (*Rechnet mit zwei Int64*) (*$GROUP=User,$CAT=User,$GROUPICON=User.png,$CATICON=User.png*)
	VAR_INPUT
		pOperand0 : BrbInt64_TYP; (*Zeiger auf die erste Int64-Struktur*)
		pOperand1 : BrbInt64_TYP; (*Zeiger auf die zweite Int64-Struktur*)
		eOperator : BrbDt64Operator_ENUM; (*Operator-Angabe (Add, Subtract, Multiply, Divide)*)
	END_VAR
END_FUNCTION
(*BigDataTypes - HelpFunctions*)

FUNCTION BrbIntegerStringAdd : DINT (*Addiert zwei Integer-Strings*) (*$GROUP=User,$CAT=User,$GROUPICON=User.png,$CATICON=User.png*)
	VAR_INPUT
		pIntegerString1 : STRING[0]; (*Zeiger auf den Anfang des ersten Integer-Strings*)
		pIntegerString2 : STRING[0]; (*Zeiger auf den Anfang des zweiten Integer-Strings*)
		nSize1 : UDINT; (*Größe des ersten Integer-Strings*)
	END_VAR
END_FUNCTION

FUNCTION BrbByteArrayAdd : DINT (*Addiert zwei Zahlen, welche als Byte-Array abgelegt sind*) (*$GROUP=User,$CAT=User,$GROUPICON=User.png,$CATICON=User.png*)
	VAR_INPUT
		pByteArray0 : REFERENCE TO USINT; (*Zeiger auf den Anfang des ersten Byte-Arrays*)
		nLength0 : UDINT; (*Länge des ersten Byte-Arrays in Byte*)
		pByteArray1 : REFERENCE TO USINT; (*Zeiger auf den Anfang des zweiten Byte-Arrays*)
		nLength1 : UDINT; (*Länge des zweiten Byte-Arrays in Byte*)
	END_VAR
END_FUNCTION

FUNCTION BrbByteArraySubtract : DINT (*Subtrahiert zwei Zahlen, welche als Byte-Array abgelegt sind*) (*$GROUP=User,$CAT=User,$GROUPICON=User.png,$CATICON=User.png*)
	VAR_INPUT
		pByteArray0 : REFERENCE TO USINT; (*Zeiger auf den Anfang des ersten Byte-Arrays*)
		nLength0 : UDINT; (*Länge des ersten Byte-Arrays in Byte*)
		pByteArray1 : REFERENCE TO USINT; (*Zeiger auf den Anfang des zweiten Byte-Arrays*)
		nLength1 : UDINT; (*Länge des zweiten Byte-Arrays in Byte*)
	END_VAR
END_FUNCTION
(*Xml*)

FUNCTION BrbXmlGetTagText : UDINT (*Gibt den Text zwischen zwei Xml-Tags zurück*)
	VAR_INPUT
		pStartTag : STRING[0]; (*Zeiger auf den Start-Tag*)
		pEndTag : STRING[0]; (*Zeiger auf den End-Tag*)
		pStart : UDINT; (*Zeiger auf den Such-Start*)
		pEnd : UDINT; (*Zeiger auf das Such-Ende*)
		pText : STRING[0]; (*Zeiger auf eine String-Variable, die das Ergebnis aufnimmt*)
		nTextSize : UDINT; (*Größe der String-Variablen*)
	END_VAR
END_FUNCTION

FUNCTION BrbXmlGetNextTag : UDINT (*Gibt die Adresse nach einem Xml-Tag zurück*)
	VAR_INPUT
		pTag : STRING[0]; (*Zeiger auf den Tag*)
		pStart : UDINT; (*Zeiger auf den Such-Start*)
		pEnd : UDINT; (*Zeiger auf das Such-Ende*)
	END_VAR
END_FUNCTION
(*Memory*)

FUNCTION BrbMemListClear : DINT (*Löscht die gesamte Liste*)
	VAR_INPUT
		pListManagement : BrbMemListManagement_Typ; (*Zeiger auf die Verwaltungs-Struktur*)
	END_VAR
END_FUNCTION

FUNCTION BrbMemListIn : DINT (*Fügt einen Eintrag an bestimmter Stelle in der Liste ein*)
	VAR_INPUT
		pListManagement : BrbMemListManagement_Typ; (*Zeiger auf die Verwaltungs-Struktur*)
		nIndex : UDINT; (*Index des Eintrags*)
		pNewEntry : UDINT; (*Zeiger auf die Daten des Eintrags*)
	END_VAR
END_FUNCTION

FUNCTION BrbMemListOut : DINT (*Holt einen bestimmten Eintrag und löscht ihn aus der Liste*)
	VAR_INPUT
		pListManagement : BrbMemListManagement_Typ; (*Zeiger auf die Verwaltungs-Struktur*)
		nIndex : UDINT; (*Index des Eintrags*)
		pListEntry : UDINT; (*Zeiger auf die Daten des Eintrags*)
	END_VAR
END_FUNCTION

FUNCTION BrbMemListGetEntry : DINT (*Holt einen bestimmten Eintrag aus der Liste*)
	VAR_INPUT
		pListManagement : BrbMemListManagement_Typ; (*Zeiger auf die Verwaltungs-Struktur*)
		nIndex : UDINT; (*Index des Eintrags*)
		pListEntry : UDINT; (*Zeiger auf die Daten des Eintrags*)
	END_VAR
END_FUNCTION

FUNCTION BrbFifoIn : DINT (*Fügt einen neuen Eintrag an der letzten Stelle hinzu*)
	VAR_INPUT
		pListManagement : BrbMemListManagement_Typ; (*Zeiger auf die Verwaltungs-Struktur*)
		pNewEntry : UDINT; (*Zeiger auf die Daten des Eintrags*)
	END_VAR
END_FUNCTION

FUNCTION BrbFifoOut : DINT (*Gibt den Eintrag an erster Stelle zurück und löscht ihn aus der Liste*)
	VAR_INPUT
		pListManagement : BrbMemListManagement_Typ; (*Zeiger auf die Verwaltungs-Struktur*)
		pListEntry : UDINT; (*Zeiger auf die Daten des Eintrags*)
	END_VAR
END_FUNCTION

FUNCTION BrbLifoIn : DINT (*Fügt einen neuen Eintrag an der letzten Stelle hinzu*)
	VAR_INPUT
		pListManagement : BrbMemListManagement_Typ; (*Zeiger auf die Verwaltungs-Struktur*)
		pNewEntry : UDINT; (*Zeiger auf die Daten des Eintrags*)
	END_VAR
END_FUNCTION

FUNCTION BrbLifoOut : DINT (*Gibt den Eintrag an letzter Stelle zurück und löscht ihn aus der Liste*)
	VAR_INPUT
		pListManagement : BrbMemListManagement_Typ; (*Zeiger auf die Verwaltungs-Struktur*)
		pListEntry : UDINT; (*Zeiger auf die Daten des Eintrags*)
	END_VAR
END_FUNCTION

FUNCTION BrbGetBitUdint : BOOL (*Liest ein Bit aus einem Udint*)
	VAR_INPUT
		nValue : UDINT; (*Udint-Wert*)
		nBitNumber : UINT; (*Nummer des Bits (0..31)*)
	END_VAR
END_FUNCTION

FUNCTION BrbSetBitUdint : BOOL (*Setzt oder löscht ein Bit in einem Udint*)
	VAR_INPUT
		pValue : REFERENCE TO UDINT; (*Zeiger auf einen Udint-Wert*)
		nBitNumber : UINT; (*Nummer des Bits (0..31)*)
		bBit : BOOL; (*0=Löschen, 1=Setzen*)
	END_VAR
END_FUNCTION

FUNCTION BrbGetBitMaskUdint : BOOL (*Liest eine Bitmaske aus einem Udint*)
	VAR_INPUT
		nValue : UDINT; (*Udint-Wert*)
		nBitMask : UDINT; (*Bit-Maske*)
	END_VAR
END_FUNCTION

FUNCTION BrbSetBitMaskUdint : BOOL (*Setzt oder löscht eine Bitmaske in einem Udint*)
	VAR_INPUT
		pValue : REFERENCE TO UDINT; (*Zeiger auf einen Udint-Wert*)
		nBitMask : UDINT; (*Bit-Maske*)
		bSet : BOOL; (*0=Löschen, 1=Setzen*)
	END_VAR
END_FUNCTION

FUNCTION BrbGetBitUint : BOOL (*Liest ein Bit aus einem Uint*)
	VAR_INPUT
		nValue : UINT; (*Uint-Wert*)
		nBitNumber : UINT; (*Nummer des Bits (0..15)*)
	END_VAR
END_FUNCTION

FUNCTION BrbSetBitUint : BOOL (*Setzt oder löscht ein Bit in einem Uint*)
	VAR_INPUT
		pValue : REFERENCE TO UINT; (*Zeiger auf einen Uint-Wert*)
		nBitNumber : UINT; (*Nummer des Bits (0..15)*)
		bBit : BOOL; (*0=Löschen, 1=Setzen*)
	END_VAR
END_FUNCTION

FUNCTION BrbGetBitMaskUint : BOOL (*Liest eine Bitmaske aus einem Uint*)
	VAR_INPUT
		nValue : UINT; (*Uint-Wert*)
		nBitMask : UINT; (*Bit-Maske*)
	END_VAR
END_FUNCTION

FUNCTION BrbSetBitMaskUint : BOOL (*Setzt oder löscht eine Bitmaske in einem Uint*)
	VAR_INPUT
		pValue : REFERENCE TO UINT; (*Zeiger auf einen Uint-Wert*)
		nBitMask : UINT; (*Bit-Maske*)
		bSet : BOOL; (*0=Löschen, 1=Setzen*)
	END_VAR
END_FUNCTION

FUNCTION BrbGetBitUsint : BOOL (*Liest ein Bit aus einem Usint*)
	VAR_INPUT
		nValue : USINT; (*Usint-Wert*)
		nBitNumber : UINT; (*Nummer des Bits (0..7)*)
	END_VAR
END_FUNCTION

FUNCTION BrbSetBitUsint : BOOL (*Setzt ein Bit in einem Usint*)
	VAR_INPUT
		pValue : REFERENCE TO USINT; (*Zeiger auf einen Usint-Wert*)
		nBitNumber : UINT; (*Nummer des Bits (0..7)*)
		bBit : BOOL; (*0=Löschen, 1=Setzen*)
	END_VAR
END_FUNCTION

FUNCTION BrbGetBitMaskUsint : BOOL (*Liest eine Bitmaske aus einem Usint*)
	VAR_INPUT
		nValue : USINT; (*Usint-Wert*)
		nBitMask : USINT; (*Bit-Maske*)
	END_VAR
END_FUNCTION

FUNCTION BrbSetBitMaskUsint : BOOL (*Setzt oder löscht eine Bitmaske in einem Usint*)
	VAR_INPUT
		pValue : REFERENCE TO USINT; (*Zeiger auf einen Usint-Wert*)
		nBitMask : USINT; (*Bit-Maske*)
		bSet : BOOL; (*0=Löschen, 1=Setzen*)
	END_VAR
END_FUNCTION

FUNCTION BrbGetByteArrayBit : BOOL (*Gibt ein Bit eines bitcodierten Byte-Arrays zurück*) (*$GROUP=User,$CAT=User,$GROUPICON=User.png,$CATICON=User.png*)
	VAR_INPUT
		pByteArray : UDINT; (*Zeiger auf das Byte-Array*)
		nIndexMax : UDINT; (*Maximaler Index des Byte-Arrays*)
		nBitNumber : UDINT; (*Nummer der Bits (0..n)*)
	END_VAR
END_FUNCTION

FUNCTION BrbSetByteArrayBit : BOOL (*Setzt ein Bit in einem bitcodierten Byte-Array*) (*$GROUP=User,$CAT=User,$GROUPICON=User.png,$CATICON=User.png*)
	VAR_INPUT
		pByteArray : UDINT; (*Zeiger auf das Byte-Array*)
		nIndexMax : UDINT; (*Maximaler Index des Byte-Arrays*)
		nBitNumber : UDINT; (*Nummer der Bits (0..n)*)
		bBit : BOOL; (*Zu setzender Wert*)
	END_VAR
END_FUNCTION

FUNCTION BrbSetByteArrayBits : BOOL (*Setzte Bits in einem bitcodierten Byte-Array*) (*$GROUP=User,$CAT=User,$GROUPICON=User.png,$CATICON=User.png*)
	VAR_INPUT
		pByteArray : UDINT; (*Zeiger auf das Byte-Array*)
		nIndexMax : UDINT; (*Maximaler Index des Byte-Arrays*)
		nBitNumberFrom : UDINT; (*Start-Nummer der Bits (0..n)*)
		nBitNumberTo : UDINT; (*End-Nummer der Bits (0..n)*)
		bBit : BOOL; (*Zu setzender Wert für jedes Bit*)
	END_VAR
END_FUNCTION
(*Math*)

FUNCTION BrbAbsReal : REAL (*Gibt den absoluten Wert zurück*) (*$GROUP=User,$CAT=User,$GROUPICON=User.png,$CATICON=User.png*)
	VAR_INPUT
		rValue : REAL; (*Wert*)
	END_VAR
END_FUNCTION

FUNCTION BrbAbsLReal : LREAL (*Gibt den absoluten Wert zurück*) (*$GROUP=User,$CAT=User,$GROUPICON=User.png,$CATICON=User.png*)
	VAR_INPUT
		rValue : LREAL; (*Wert*)
	END_VAR
END_FUNCTION

FUNCTION BrbIsNearlyZeroReal : BOOL (*Gibt zurück, ob ein REAL-Wert annähernd 0 ist*) (*$GROUP=User,$CAT=User,$GROUPICON=User.png,$CATICON=User.png*)
	VAR_INPUT
		rValue : REAL; (*Wert*)
		rTolerance : REAL; (*Grenz-Toleranz*)
	END_VAR
END_FUNCTION

FUNCTION BrbIsNearlyZeroLReal : BOOL (*Gibt zurück, ob ein LREAL-Wert annähernd 0 ist*) (*$GROUP=User,$CAT=User,$GROUPICON=User.png,$CATICON=User.png*)
	VAR_INPUT
		rValue : LREAL; (*Wert*)
		rTolerance : LREAL; (*Grenz-Toleranz*)
	END_VAR
END_FUNCTION

FUNCTION BrbCompareReal : INT (*Vergleicht zwei REAL-Werte*) (*$GROUP=User,$CAT=User,$GROUPICON=User.png,$CATICON=User.png*)
	VAR_INPUT
		rValue1 : REAL; (*1. Wert*)
		rValue2 : REAL; (*2. Wert*)
	END_VAR
END_FUNCTION

FUNCTION BrbCompareLReal : INT (*Vergleicht zwei LREAL-Werte*) (*$GROUP=User,$CAT=User,$GROUPICON=User.png,$CATICON=User.png*)
	VAR_INPUT
		rValue1 : LREAL; (*1. Wert*)
		rValue2 : LREAL; (*2. Wert*)
	END_VAR
END_FUNCTION

FUNCTION BrbIsWithinRangeDint : BOOL (*Gibt zurück, ob sich ein Wert innerhalb eines Bereichs befindet*) (*$GROUP=User,$CAT=User,$GROUPICON=User.png,$CATICON=User.png*)
	VAR_INPUT
		nValue : DINT; (*Wert*)
		nRangeMin : DINT; (*Untere Grenze*)
		nRangeMax : DINT; (*Obere Grenze*)
		nTolerance : DINT; (*Grenz-Toleranz*)
	END_VAR
END_FUNCTION

FUNCTION BrbIsWithinRangeUdint : BOOL (*Gibt zurück, ob sich ein Wert innerhalb eines Bereichs befindet*) (*$GROUP=User,$CAT=User,$GROUPICON=User.png,$CATICON=User.png*)
	VAR_INPUT
		nValue : UDINT; (*Wert*)
		nRangeMin : UDINT; (*Untere Grenze*)
		nRangeMax : UDINT; (*Obere Grenze*)
		nTolerance : UDINT; (*Grenz-Toleranz*)
	END_VAR
END_FUNCTION

FUNCTION BrbIsWithinRangeReal : BOOL (*Gibt zurück, ob sich ein Wert innerhalb eines Bereichs befindet*) (*$GROUP=User,$CAT=User,$GROUPICON=User.png,$CATICON=User.png*)
	VAR_INPUT
		rValue : REAL; (*Wert*)
		rRangeMin : REAL; (*Untere Grenze*)
		rRangeMax : REAL; (*Obere Grenze*)
		rTolerance : REAL; (*Grenz-Toleranz*)
	END_VAR
END_FUNCTION

FUNCTION BrbIsWithinRangeLReal : BOOL (*Gibt zurück, ob sich ein Wert innerhalb eines Bereichs befindet*) (*$GROUP=User,$CAT=User,$GROUPICON=User.png,$CATICON=User.png*)
	VAR_INPUT
		rValue : LREAL; (*Wert*)
		rRangeMin : LREAL; (*Untere Grenze*)
		rRangeMax : LREAL; (*Obere Grenze*)
		rTolerance : LREAL; (*Grenz-Toleranz*)
	END_VAR
END_FUNCTION

FUNCTION BrbGetAngleRad : REAL (*Rechnet einen Winkel von Grad ins Bogenmass um*)
	VAR_INPUT
		rAngleDeg : REAL; (*Winkel in Grad*)
	END_VAR
END_FUNCTION

FUNCTION BrbGetAngleDeg : REAL (*Rechnet einen Winkel vom Bogenmass in Grad um*)
	VAR_INPUT
		rAngleRad : REAL; (*Winkel im Bogenmass*)
	END_VAR
END_FUNCTION

FUNCTION BrbNormalizeAngleRad : REAL (*Normalisiert einen Bogenmass-Winkel in den Bereich 0..2Pi*)
	VAR_INPUT
		rAngleRad : REAL; (*Winkel im Bogenmass*)
	END_VAR
END_FUNCTION

FUNCTION BrbNormalizeAngleDeg : REAL (*Normalisiert einen Grad-Winkel in den Bereich 0..360°*)
	VAR_INPUT
		rAngleDeg : REAL; (*Winkel in Grad*)
		bKeep360 : USINT; (*Genau 360.0° werden nicht zu 0.0°*)
	END_VAR
END_FUNCTION

FUNCTION BrbIsWithinRangeAngle : BOOL (*Gibt zurück, ob sich ein Winkel innerhalb eines Bereichs befindet*) (*$GROUP=User,$CAT=User,$GROUPICON=User.png,$CATICON=User.png*)
	VAR_INPUT
		rAngleAct : LREAL; (*Zu prüfender Winkel*)
		rAngleStart : LREAL; (*Start-Winkel des Bereichs*)
		rAngleEnd : LREAL; (*End-Winkel des Bereichs*)
	END_VAR
END_FUNCTION

FUNCTION BrbDetectAngleTransition : BOOL (*Erkennt den Übergang einer bestimmten Position bei einer 360°-Rundachse*) (*$GROUP=User,$CAT=User,$GROUPICON=User.png,$CATICON=User.png*)
	VAR_INPUT
		rTransPosition : LREAL; (*Zu erkennende Übergangs-Position [°]*)
		bDirection : BOOL; (*Richtung: 0=Negativ; 1=Positiv*)
		rPosAct : LREAL; (*Aktuelle Rundachs-Position [0°..360°]*)
		rPosOld : LREAL; (*Alte Rundachs-Position [0°..360°] vom vorigen Task-Zyklus*)
	END_VAR
END_FUNCTION

FUNCTION BrbGetDistance2d : LREAL (*Gibt die Distanz zwischen zwei Punkten im 2-dimensionalen Raum zurück*) (*$GROUP=User,$CAT=User,$GROUPICON=User.png,$CATICON=User.png*)
	VAR_INPUT
		rX1 : LREAL; (*X-Koordinate des 1. Punkts*)
		rY1 : LREAL; (*Y-Koordinate des 1. Punkts*)
		rX2 : LREAL; (*X-Koordinate des 2. Punkts*)
		rY2 : LREAL; (*Y-Koordinate des 2. Punkts*)
	END_VAR
END_FUNCTION

FUNCTION BrbRoundDint : DINT (*Rundet einen Dint*)
	VAR_INPUT
		nValue : DINT; (*Zu rundendet Wert*)
		eRound : BrbRound_ENUM; (*Rundungstyp*)
		nDigits : USINT; (*Stelle, auf die gerundet wird*)
	END_VAR
END_FUNCTION

FUNCTION BrbScaleLReal : LREAL (*Skaliert ein analoges Signal linear*) (*$GROUP=User*)
	VAR_INPUT
		rRaw : LREAL; (*Rohwert*)
		rRawMin : LREAL; (*Minimaler Rohwert*)
		rRawMax : LREAL; (*Maximaler Rohwert*)
		rScaledMin : LREAL; (*Minimaler skalierter Wert*)
		rScaledMax : LREAL; (*Maximaler skalierter Wert*)
		rFactor : LREAL; (*Umrechnungs-Faktor*)
		rOffset : LREAL; (*Umrechnungs-Offset*)
	END_VAR
END_FUNCTION

FUNCTION BrbScaleAnalogInput : REAL (*Skaliert ein analoges Eingangssignal linear auf einen Einheitswert*) (*$GROUP=User*)
	VAR_INPUT
		nRaw : INT; (*Rohwert*)
		nRawMin : INT; (*Minimaler Rohwert*)
		nRawMax : INT; (*Maximaler Rohwert*)
		rScaledMin : REAL; (*Minimaler skalierter Wert*)
		rScaledMax : REAL; (*Maximaler skalierter Wert*)
		rFactor : REAL; (*Umrechnungs-Faktor*)
		rOffset : REAL; (*Umrechnungs-Offset*)
	END_VAR
END_FUNCTION

FUNCTION BrbScaleAnalogOutput : INT (*Skaliert ein analoges Ausgangssignal von einem Einheitswert*) (*$GROUP=User*)
	VAR_INPUT
		rScaled : REAL; (*Einheitswert*)
		nRawMin : INT; (*Minimaler Rohwert*)
		nRawMax : INT; (*Maximaler Rohwert*)
		rScaledMin : REAL; (*Minimaler skalierter Wert*)
		rScaledMax : REAL; (*Maximaler skalierter Wert*)
		rFactor : REAL; (*Umrechnungs-Faktor*)
		rOffset : REAL; (*Umrechnungs-Offset*)
	END_VAR
END_FUNCTION
(*Random*)

FUNCTION BrbGetRandomPercent : REAL (*Erzeugt eine Zufallszahl zwischen 0.0 und 1.0*)
END_FUNCTION

FUNCTION BrbGetRandomBool : BOOL (*Erzeugt einen boolschen Zufallswert*)
END_FUNCTION

FUNCTION BrbGetRandomUdint : UDINT (*Erzeugt eine Zufallszahl zwischen nMin und nMax*)
	VAR_INPUT
		nMin : UDINT; (*Minimaler Zahlenwert*)
		nMax : UDINT; (*Maximaler Zahlenwert*)
	END_VAR
END_FUNCTION

FUNCTION BrbGetRandomDint : DINT (*Erzeugt eine Zufallszahl zwischen nMin und nMax*)
	VAR_INPUT
		nMin : DINT; (*Minimaler Zahlenwert*)
		nMax : DINT; (*Maximaler Zahlenwert*)
	END_VAR
END_FUNCTION

FUNCTION BrbGetRandomText : UDINT (*Erzeugt einen Zufallstext mit bestimmter Länge (nur Zahlen, Groß- und Kleinbuchstaben)*) (*$GROUP=User,$CAT=User,$GROUPICON=User.png,$CATICON=User.png*)
	VAR_INPUT
		pText : STRING[0]; (*Zeiger auf den Text*)
		nTextSize : UDINT; (*Größe der String-Variablen*)
		nTextLength : UDINT; (*Länge der zu erstellenden Textes*)
	END_VAR
END_FUNCTION

FUNCTION BrbGetRandomString : UDINT (*Erzeugt einen Zufallstext mit bestimmter Länge aus einer Zeichenblockauswahl*) (*$GROUP=User,$CAT=User,$GROUPICON=User.png,$CATICON=User.png*)
	VAR_INPUT
		pText : STRING[0]; (*Zeiger auf den Text*)
		nTextSize : UDINT; (*Größe der String-Variablen*)
		nTextLength : UDINT; (*Länge der zu erstellenden Textes*)
		eSelection : BrbRandomString_ENUM; (*Auswahl*)
	END_VAR
END_FUNCTION

FUNCTION BrbGetRandomStringExt : UDINT (*Erzeugt einen Zufallstext mit bestimmter Länge aus einer Zeichenauswahl*) (*$GROUP=User,$CAT=User,$GROUPICON=User.png,$CATICON=User.png*)
	VAR_INPUT
		pText : STRING[0]; (*Zeiger auf den Text*)
		nTextSize : UDINT; (*Größe der String-Variablen*)
		nTextLength : UDINT; (*Länge der zu erstellenden Textes*)
		pSelection : STRING[0]; (*Zeiger auf den Auswahl-Text*)
	END_VAR
END_FUNCTION
(*IpAndSubnet*)

FUNCTION BrbIpToNumericalArray : UINT (*Wandelt eine textuelle Ip-Adresse in ein USINT-Array*) (*$GROUP=User,$CAT=User,$GROUPICON=User.png,$CATICON=User.png*)
	VAR_INPUT
		pIp : STRING[0]; (*Zeiger auf den Ip-Adress-Text*)
		pUsintArray : UDINT; (*Zeiger auf USINT-Array mit 4 Elementen*)
	END_VAR
END_FUNCTION

FUNCTION BrbCheckIpAddress : BOOL (*Prüft eine Ip-Adresse und berichtigt sie gegebenenfalls*)
	VAR_INPUT
		pIpAddress : STRING[0]; (*Zeiger auf den Ip-Adress-Text*)
	END_VAR
END_FUNCTION

FUNCTION BrbCheckSubnet : BOOL (*Prüft eine Subnet-Angabe auf Gültigkeit*) (*$GROUP=User,$CAT=User,$GROUPICON=User.png,$CATICON=User.png*)
	VAR_INPUT
		pSubnet : STRING[0]; (*Zeiger auf den Subnet-Text*)
	END_VAR
END_FUNCTION

FUNCTION BrbGetIpAddressType : BrbIpAdrType_ENUM (*Gibt den Typen einer Ip-Adresse zurück (Netzwerk-oder Broadcast-Adresse)*) (*$GROUP=User,$CAT=User,$GROUPICON=User.png,$CATICON=User.png*)
	VAR_INPUT
		pIp : STRING[0]; (*Zeiger auf den Ip-Adress-Text*)
		pSubnet : STRING[0]; (*Zeiger auf den Subnet-Text*)
	END_VAR
END_FUNCTION

FUNCTION BrbCheckIpEqualSubnet : BOOL (*Prüft, ob zwei Ip-Adressen im selben Subnet sind*) (*$GROUP=User,$CAT=User,$GROUPICON=User.png,$CATICON=User.png*)
	VAR_INPUT
		pIp1 : STRING[0]; (*Zeiger auf den ersten Ip-Adress-Text*)
		pSubnet1 : STRING[0]; (*Zeiger auf den ersten Subnet-Text*)
		pIp2 : STRING[0]; (*Zeiger auf den zweiten Ip-Adress-Text*)
		pSubnet2 : STRING[0]; (*Zeiger auf den zweiten Subnet-Text*)
	END_VAR
END_FUNCTION
(*Additional*)

{REDUND_UNREPLICABLE} FUNCTION_BLOCK BrbDebounceInput (*Entprellt einen Eingang*)
	VAR_INPUT
		bInput : {REDUND_UNREPLICABLE} BOOL; (*Zu entprellender Eingang*)
		nDebounceTime : {REDUND_UNREPLICABLE} UDINT; (*Entprell-Zeit [ms]*)
	END_VAR
	VAR_OUTPUT
		bOutput : {REDUND_UNREPLICABLE} BOOL; (*Entprellter Eingang*)
	END_VAR
	VAR
		fbDebounce : {REDUND_UNREPLICABLE} TON; (*Interner Fub*)
	END_VAR
END_FUNCTION_BLOCK

FUNCTION BrbGetStructMemberOffset : UINT (*Gibt den Offset eines Struktur-Members zurück*)
	VAR_INPUT
		pStructName : STRING[0]; (*Zeiger auf den Namen der Struktur-Instanz*)
		pMemberName : STRING[0]; (*Zeiger auf dem Namen des Struktur-Elements*)
		pOffset : REFERENCE TO UDINT; (*Zeiger auf den Offset*)
	END_VAR
END_FUNCTION

FUNCTION BrbGetCompilerVersion : UINT (*Gibt die Version des verwendeten GCC-Compilers zurück*) (*$GROUP=User,$CAT=User,$GROUPICON=User.png,$CATICON=User.png*)
	VAR_INPUT
		pCompilerVersion : BrbCompilerVersion_TYP; (*Zeiger auf die Version-Struktur*)
	END_VAR
END_FUNCTION
```
